      ELSIF (_Mover.NcToPlc.ModuloActPos > stGearData.rModuloSyncPosSlave + stMoveData.rDelta)
      THEN
        _nErrorId             := 667;
        _eState               := E_PROGRESS.PROGRESS_ERROR;
      END_IF
    END_IF
END_CASE
//-----------------------------------------------------------------------------
//-----------------------------------------------------------------------------
CASE _eState
OF
  E_PROGRESS.PROGRESS_BUSY:
    _eState                   := E_PROGRESS.PROGRESS_PREPARE;

    _fbPower.Override         := stMoveData.rOverride;

    _fbGearInPosCa(
        Master                := _Master, 
        Slave                 := _Mover, 
        Execute               := FALSE, 
        ContinuousUpdate      := TRUE, 
        RatioNumerator        := stGearData.rGearNumerator, 
        RatioDenumerator      := stGearData.iGearDenumerator, 

        MasterSyncPosition    := _Master.NcToPlc.ActPos 
                               + stGearData.rDeltaToMasterPos,                            // absolute position

        SlaveSyncPosition     := ABS(_Mover.NcToPlc.ModuloActTurns)*_RailLength
                               + stGearData.rModuloSyncPosSlave,                          // absolute position

        SyncStrategy          := Tc3_Mc3Definitions.MC_SYNC_STRATEGY.mcSyncStrategySlow,  // minimal movement with this strategy 
        SyncMode              := Tc3_Mc3Definitions.MC_SYNC_MODE.mcSyncModeNonModulo,     // all positions as absolute value
        MasterStartDistance   := stGearData.rMasterStartDistance,                         // if <> 0 --> master has to move before this fb does anything
        Velocity              := stMoveData.rVelo, 
        Acceleration          := stMoveData.rAcc, 
        Deceleration          := stMoveData.rAcc, 
        Jerk                  := stMoveData.rJerk, 
        Gap                   := stMoveData.rGap, 
        BufferMode            := Tc3_Mc3Definitions.MC_BUFFER_MODE.mcAborting);
END_CASE
//-----------------------------------------------------------------------------
//-----------------------------------------------------------------------------
CASE _eState
OF
  E_PROGRESS.PROGRESS_PREPARE:
    _fbGearInPosCa(
        Master                := _Master, 
        Slave                 := _Mover, 
        Execute               := TRUE, 
        ContinuousUpdate      := TRUE);

    IF _fbGearInPosCa.Error
    THEN
      _nErrorId               := _fbGearInPosCa.ErrorId;
      _eState                 := E_PROGRESS.PROGRESS_ERROR;

    ELSIF _fbGearInPosCa.CommandAborted
    THEN
      _eState                 := E_PROGRESS.PROGRESS_OCCUPIED;

    ELSIF _fbGearInPosCa.InSync
    THEN
      _eState                 := E_PROGRESS.PROGRESS_DONE;
    END_IF
END_CASE
//-----------------------------------------------------------------------------
//-----------------------------------------------------------------------------
CASE _eState
OF
  E_PROGRESS.PROGRESS_ERROR,
  E_PROGRESS.PROGRESS_DONE:
    _stInfo.nErrorId          := _nErrorId;
    _fbGearInPosCa(
        Master                := _Master, 
        Slave                 := _Mover, 
        Execute               := FALSE, 
        ContinuousUpdate      := TRUE);
END_CASE
//-----------------------------------------------------------------------------
//-----------------------------------------------------------------------------

GearInPosCa                   := _eState;
END_METHOD

METHOD GearOut : E_PROGRESS
VAR_INPUT
  Execute             : BOOL;
END_VAR
VAR_INST
  _nErrorId           : UDINT;
  _eState             : E_PROGRESS;
END_VAR
IF NOT Execute THEN _eState  := E_PROGRESS.PROGRESS_INIT; END_IF 
IF NOT Check() THEN GearOut  := E_PROGRESS.PROGRESS_ERROR; RETURN; END_IF


CASE _eState
OF
  E_PROGRESS.PROGRESS_INIT:
    IF Execute
    THEN
      _nErrorId               := 0;
      _eState                 := E_PROGRESS.PROGRESS_BUSY;
    END_IF
END_CASE
//-----------------------------------------------------------------------------
//-----------------------------------------------------------------------------
CASE _eState
OF
  E_PROGRESS.PROGRESS_BUSY:
    _eState                   := E_PROGRESS.PROGRESS_PREPARE;
    _fbGearOut(
            Slave             := _Mover, 
            Execute           := FALSE);
END_CASE
//-----------------------------------------------------------------------------
//-----------------------------------------------------------------------------
CASE _eState
OF
  E_PROGRESS.PROGRESS_PREPARE:
    _fbGearOut(
            Slave             := _Mover, 
            Execute           := TRUE);

    IF _fbGearOut.Error
    THEN
      _nErrorId               := _fbGearOut.ErrorID;
      _eState                 := E_PROGRESS.PROGRESS_ERROR;

    ELSIF (_Mover.NcToPlc.CoupleState = 0)
    THEN
      _eState                 := E_PROGRESS.PROGRESS_DONE;
    END_IF
END_CASE
//-----------------------------------------------------------------------------
//-----------------------------------------------------------------------------
CASE _eState
OF
  E_PROGRESS.PROGRESS_ERROR,
  E_PROGRESS.PROGRESS_DONE:
    _stInfo.nErrorId          := _nErrorId;
    _fbGearOut(
            Slave             := _Mover, 
            Execute           := FALSE);
END_CASE
//-----------------------------------------------------------------------------
//-----------------------------------------------------------------------------

GearOut                       := _eState;
END_METHOD

METHOD Halt : E_PROGRESS
VAR_INPUT
  Execute             : BOOL;
  stMoveData          : ST_MOVE_DATA;
END_VAR
VAR_INST
  _nErrorId           : UDINT;
  _eState             : E_PROGRESS;
END_VAR
IF NOT Execute 
THEN 
	_eState := E_PROGRESS.PROGRESS_INIT; 
END_IF 
IF NOT Check() 
THEN 
	Halt := E_PROGRESS.PROGRESS_ERROR; 
	RETURN; 
END_IF


CASE _eState
OF
  E_PROGRESS.PROGRESS_INIT:
    IF Execute
    THEN
      _nErrorId               := 0;
      _eState                 := E_PROGRESS.PROGRESS_BUSY;
    END_IF
END_CASE
//-----------------------------------------------------------------------------
//-----------------------------------------------------------------------------
CASE _eState
OF
  E_PROGRESS.PROGRESS_BUSY:
    _eState                   := E_PROGRESS.PROGRESS_PREPARE;
    _fbHalt(
            Axis              := _Mover, 
            Execute           := FALSE, 
            Deceleration      := stMoveData.rAcc, 
            Jerk              := stMoveData.rJerk, 
            BufferMode        := Tc2_MC2.MC_BufferMode.MC_Aborting);
END_CASE
//-----------------------------------------------------------------------------
//-----------------------------------------------------------------------------
CASE _eState
OF
  E_PROGRESS.PROGRESS_PREPARE:
    _fbHalt(Axis              := _Mover, 
            Execute           := TRUE, 
            Deceleration      := stMoveData.rAcc, 
            Jerk              := stMoveData.rJerk, 
            BufferMode        := Tc2_MC2.MC_BufferMode.MC_Aborting);

    IF _fbHalt.Error
    THEN
      _nErrorId               := _fbHalt.ErrorID;
      _eState                 := E_PROGRESS.PROGRESS_ERROR;

    ELSIF NOT _Mover.Status.Moving
    THEN
      _eState                 := E_PROGRESS.PROGRESS_DONE;
    END_IF
END_CASE
//-----------------------------------------------------------------------------
//-----------------------------------------------------------------------------
CASE _eState
OF
  E_PROGRESS.PROGRESS_ERROR,
  E_PROGRESS.PROGRESS_DONE:
    _stInfo.nErrorId          := _nErrorId;
    _fbHalt(
            Axis              := _Mover, 
            Execute           := FALSE);
END_CASE
//-----------------------------------------------------------------------------
//-----------------------------------------------------------------------------

Halt                          := _eState;
END_METHOD

PROPERTY LastGap : REFERENCE to lreal
SET
_rLastGap REF= LastGap;
END_SET
END_PROPERTY

PROPERTY LastPosition : REFERENCE to LREAL
SET
_rLastPosition REF= LastPosition;
END_SET
END_PROPERTY

PROPERTY Master : REFERENCE to AXIS_REF
SET
_Master REF= Master;
END_SET
END_PROPERTY

PROPERTY ModuloTurn : dint
GET
ModuloTurn := _Mover.NcToPlc.ModuloSetTurns;
END_GET
END_PROPERTY

PROPERTY Mover : REFERENCE to AXIS_REF
SET
_Mover REF= Mover;
END_SET
END_PROPERTY

PROPERTY MoverInfo : REFERENCE to ST_MOVER_INFO
SET


	_stInfo ref= MoverInfo;
END_SET
END_PROPERTY

METHOD MoveToPos : E_PROGRESS
VAR_INPUT
  Execute             : BOOL;
  stMoveData          : ST_MOVE_DATA;
END_VAR
VAR_INST
  _nErrorId           : UDINT;
  _rPos               : LREAL;
  _eState             : E_PROGRESS;
END_VAR
IF NOT Execute THEN _eState  := E_PROGRESS.PROGRESS_INIT; END_IF 
IF NOT Check() THEN MoveToPos   := E_PROGRESS.PROGRESS_ERROR; RETURN; END_IF


CASE _eState
OF
  E_PROGRESS.PROGRESS_INIT:
    IF Execute
    THEN
      _nErrorId               := 0;
      _eState                 := E_PROGRESS.PROGRESS_BUSY;
    END_IF
END_CASE
//-----------------------------------------------------------------------------
//-----------------------------------------------------------------------------
CASE _eState
OF
  E_PROGRESS.PROGRESS_BUSY:
    _eState                   := E_PROGRESS.PROGRESS_PREPARE;
    _fbPower.Override         := stMoveData.rOverride;

    _rPos                     := ABS(_Mover.NcToPlc.ModuloActTurns)* _RailLength + stMoveData.rPos;


    _rLastPosition            := _rPos;
    //_rLastGap                 := stMoveData.rGap;

    _fbMoveAbs(
            Axis              := _Mover, 
            Execute           := FALSE, 
            Position          := _rPos, 
            Velocity          := stMoveData.rVelo, 
            Acceleration      := stMoveData.rAcc, 
            Deceleration      := stMoveData.rAcc, 
            Jerk              := stMoveData.rJerk, 
            BufferMode        := Tc2_MC2.MC_BufferMode.MC_Aborting);
END_CASE
//-----------------------------------------------------------------------------
//-----------------------------------------------------------------------------
CASE _eState
OF
  E_PROGRESS.PROGRESS_PREPARE:
    _fbMoveAbs(
            Axis              := _Mover, 
            Execute           := TRUE, 
            Position          := _rPos, 
            Velocity          := stMoveData.rVelo, 
            Acceleration      := stMoveData.rAcc, 
            Deceleration      := stMoveData.rAcc, 
            Jerk              := stMoveData.rJerk, 
            BufferMode        := Tc2_MC2.MC_BufferMode.MC_Aborting);

    IF _fbMoveAbs.Error
    THEN
      _nErrorId               := _fbMoveAbs.ErrorId;
      _eState                 := E_PROGRESS.PROGRESS_ERROR;

    ELSIF _fbMoveAbs.Active OR 
          _fbMoveAbs.Done
		THEN
      _eState                 := E_PROGRESS.PROGRESS_WORKING;
    END_IF
END_CASE
//-----------------------------------------------------------------------------
//-----------------------------------------------------------------------------
CASE _eState
OF
  E_PROGRESS.PROGRESS_WORKING:
    _fbMoveAbs(
          Axis              := _Mover);

    IF _fbMoveAbs.Error
    THEN
      _nErrorId             := _fbMoveAbs.ErrorId;
      _eState               := E_PROGRESS.PROGRESS_ERROR;

    ELSIF (_Mover.NcToPlc.ActPos > _fbMoveAbs.Position - stMoveData.rDelta) AND
          (_Mover.NcToPlc.ActPos < _fbMoveAbs.Position + stMoveData.rDelta)
    THEN
      IF NOT _Mover.Status.Moving
      THEN
        _eState               := E_PROGRESS.PROGRESS_DONE;
      END_IF
    END_IF
END_CASE
//-----------------------------------------------------------------------------
//-----------------------------------------------------------------------------
CASE _eState
OF
  E_PROGRESS.PROGRESS_ERROR,
  E_PROGRESS.PROGRESS_DONE:
    _stInfo.nErrorId          := _nErrorId;
    _fbMoveAbs( 
            Axis              := _Mover, 
            Execute           := FALSE);
END_CASE
//-----------------------------------------------------------------------------
//-----------------------------------------------------------------------------

MoveToPos                   := _eState;
END_METHOD

METHOD MoveToPosCa : E_PROGRESS
VAR_INPUT
  Execute             : BOOL;
  stMoveData          : ST_MOVE_DATA;
END_VAR
VAR_INST
  _nErrorId           : UDINT;
  _rPos               : LREAL;
  _eState             : E_PROGRESS;
END_VAR
IF NOT Execute THEN _eState  := E_PROGRESS.PROGRESS_INIT; END_IF 
IF NOT Check() THEN MoveToPosCa   := E_PROGRESS.PROGRESS_ERROR; RETURN; END_IF


CASE _eState
OF
  E_PROGRESS.PROGRESS_INIT:
    IF Execute
    THEN
      _nErrorId               := 0;
      _eState                 := E_PROGRESS.PROGRESS_BUSY;
    END_IF
END_CASE
//-----------------------------------------------------------------------------
//-----------------------------------------------------------------------------
CASE _eState
OF
  E_PROGRESS.PROGRESS_BUSY:
    _eState                   := E_PROGRESS.PROGRESS_PREPARE;
    _fbPower.Override         := stMoveData.rOverride;

    _rPos                     := ABS(_Mover.NcToPlc.ModuloActTurns)* _RailLength + stMoveData.rPos;


    _rLastPosition            := _rPos;
    _rLastGap                 := stMoveData.rGap;

    _fbMoveAbsCa( 
            Axis              := _Mover, 
            Execute           := FALSE, 
            ContinuousUpdate  := TRUE, 
            Position          := _rPos,
            Velocity          := stMoveData.rVelo, 
            Acceleration      := stMoveData.rAcc, 
            Deceleration      := stMoveData.rAcc, 
            Jerk              := stMoveData.rJerk, 
            Gap               := stMoveData.rGap, 
            BufferMode        := Tc3_Mc3Definitions.MC_BUFFER_MODE.mcAborting);
END_CASE
//-----------------------------------------------------------------------------
//-----------------------------------------------------------------------------
CASE _eState
OF
  E_PROGRESS.PROGRESS_PREPARE:
    _fbMoveAbsCa( 
            Axis              := _Mover, 
            Execute           := TRUE, 
            ContinuousUpdate  := TRUE, 
            Position          := _rPos,
            Velocity          := stMoveData.rVelo, 
            Acceleration      := stMoveData.rAcc, 
            Deceleration      := stMoveData.rAcc, 
            Jerk              := stMoveData.rJerk, 
            Gap               := stMoveData.rGap, 
            BufferMode        := Tc3_Mc3Definitions.MC_BUFFER_MODE.mcAborting);

    IF _fbMoveAbsCa.Error
    THEN
      _nErrorId               := _fbMoveAbsCa.ErrorId;
      _eState                 := E_PROGRESS.PROGRESS_ERROR;

    ELSIF _fbMoveAbsCa.Active OR 
          _fbMoveAbsCa.Done
		THEN
      _eState                 := E_PROGRESS.PROGRESS_WORKING;
    END_IF
END_CASE
//-----------------------------------------------------------------------------
//-----------------------------------------------------------------------------
CASE _eState
OF
  E_PROGRESS.PROGRESS_WORKING:
    _fbMoveAbsCa(
          Axis              := _Mover);

    IF _fbMoveAbsCa.Error
    THEN
      _nErrorId             := _fbMoveAbsCa.ErrorId;
      _eState               := E_PROGRESS.PROGRESS_ERROR;

    ELSIF (_Mover.NcToPlc.ActPos > _fbMoveAbsCa.Position - stMoveData.rDelta) AND
          (_Mover.NcToPlc.ActPos < _fbMoveAbsCa.Position + stMoveData.rDelta)
    THEN
      IF NOT _Mover.Status.Moving
      THEN
        _eState               := E_PROGRESS.PROGRESS_DONE;
      END_IF
    END_IF
END_CASE
//-----------------------------------------------------------------------------
//-----------------------------------------------------------------------------
CASE _eState
OF
  E_PROGRESS.PROGRESS_ERROR,
  E_PROGRESS.PROGRESS_DONE:
    _stInfo.nErrorId          := _nErrorId;
    _fbMoveAbsCa( 
            Axis              := _Mover, 
            Execute           := FALSE);
END_CASE
//-----------------------------------------------------------------------------
//-----------------------------------------------------------------------------

MoveToPosCa                   := _eState;
END_METHOD

PROPERTY RailLength : LREAL
GET
RailLength := _RailLength;
END_GET
SET
_RailLength := RailLength;
END_SET
END_PROPERTY

METHOD Reset : E_PROGRESS
VAR_INPUT
  Execute             : BOOL;
END_VAR
VAR_INST
  _nErrorId           : UDINT;
  _eState             : E_PROGRESS;
END_VAR
IF NOT Execute THEN _eState  := E_PROGRESS.PROGRESS_INIT; END_IF 
IF NOT Check() THEN Reset    := E_PROGRESS.PROGRESS_ERROR; RETURN; END_IF


CASE _eState
OF
  E_PROGRESS.PROGRESS_INIT:
    IF Execute
    THEN
      _stInfo.nErrorId        :=
      _nErrorId               := 0;
      _eState                 := E_PROGRESS.PROGRESS_BUSY;
    END_IF
END_CASE
//-----------------------------------------------------------------------------
//-----------------------------------------------------------------------------
CASE _eState
OF
  E_PROGRESS.PROGRESS_BUSY:
    _eState                   := E_PROGRESS.PROGRESS_PREPARE;
    _fbReset(
            Axis              := _Mover, 
            Execute           := FALSE);
END_CASE
//-----------------------------------------------------------------------------
//-----------------------------------------------------------------------------
CASE _eState
OF
  E_PROGRESS.PROGRESS_PREPARE:
    _fbReset(
            Axis              := _Mover, 
            Execute           := TRUE);

    IF _fbReset.Error
    THEN
      _nErrorId               := _fbReset.ErrorID;
      _eState                 := E_PROGRESS.PROGRESS_ERROR;

    ELSIF NOT _Mover.Status.Moving
    THEN
      _eState                 := E_PROGRESS.PROGRESS_DONE;
    END_IF
END_CASE
//-----------------------------------------------------------------------------
//-----------------------------------------------------------------------------
CASE _eState
OF
  E_PROGRESS.PROGRESS_ERROR,
  E_PROGRESS.PROGRESS_DONE:
    _stInfo.nErrorId          := _nErrorId;
    _fbReset(
            Axis              := _Mover, 
            Execute           := FALSE);
			
	_bError := FALSE;		
END_CASE
//-----------------------------------------------------------------------------
//-----------------------------------------------------------------------------

Reset                         := _eState;
END_METHOD

METHOD SendToAbsPosCa : E_PROGRESS
VAR_INPUT
  Execute             : BOOL;
  stMoveData          : ST_MOVE_DATA;
END_VAR
VAR_INST
  _nErrorId           : UDINT;
  _rPos               : LREAL;
  _rStart             : LREAL;
  _eState             : E_PROGRESS;
END_VAR
IF NOT Execute THEN _eState  := E_PROGRESS.PROGRESS_INIT; END_IF 
IF NOT Check() THEN SendToAbsPosCa   := E_PROGRESS.PROGRESS_ERROR; RETURN; END_IF


CASE _eState
OF
  E_PROGRESS.PROGRESS_INIT:
    IF Execute
    THEN
      _nErrorId               := 0;
      _rStart                 := _Mover.NcToPlc.ActPos;

      _eState                 := E_PROGRESS.PROGRESS_BUSY;
    END_IF
END_CASE
//-----------------------------------------------------------------------------
//-----------------------------------------------------------------------------
CASE _eState
OF
  E_PROGRESS.PROGRESS_BUSY:
    _eState                   := E_PROGRESS.PROGRESS_PREPARE;
    _fbPower.Override         := stMoveData.rOverride;

    _rPos                     := stMoveData.rPos;
	
    _rLastPosition            := _rPos;
    _rLastGap                 := stMoveData.rGap;

    _fbMoveAbsCa( 
            Axis              := _Mover, 
            Execute           := FALSE, 
            ContinuousUpdate  := TRUE, 
            Position          := _rPos,
            Velocity          := stMoveData.rVelo, 
            Acceleration      := stMoveData.rAcc, 
            Deceleration      := stMoveData.rAcc, 
            Jerk              := stMoveData.rJerk, 
            Gap               := stMoveData.rGap, 
            BufferMode        := Tc3_Mc3Definitions.MC_BUFFER_MODE.mcAborting);
END_CASE
//-----------------------------------------------------------------------------
//-----------------------------------------------------------------------------
CASE _eState
OF
  E_PROGRESS.PROGRESS_PREPARE:
    _fbMoveAbsCa( 
            Axis              := _Mover, 
            Execute           := TRUE, 
            ContinuousUpdate  := TRUE, 
            Position          := _rPos,
            Velocity          := stMoveData.rVelo, 
            Acceleration      := stMoveData.rAcc, 
            Deceleration      := stMoveData.rAcc, 
            Jerk              := stMoveData.rJerk, 
            Gap               := stMoveData.rGap, 
            BufferMode        := Tc3_Mc3Definitions.MC_BUFFER_MODE.mcAborting);

    IF _fbMoveAbsCa.Error
    THEN
      _nErrorId               := _fbMoveAbsCa.ErrorId;
      _eState                 := E_PROGRESS.PROGRESS_ERROR;

    ELSIF _fbMoveAbsCa.Active
    THEN
      _eState                 := E_PROGRESS.PROGRESS_WORKING;
    END_IF
END_CASE
//-----------------------------------------------------------------------------
//-----------------------------------------------------------------------------
CASE _eState
OF
  E_PROGRESS.PROGRESS_WORKING:
    _fbMoveAbsCa(
            Axis              := _Mover);

    IF _fbMoveAbsCa.Error
    THEN
      _nErrorId               := _fbMoveAbsCa.ErrorId;
      _eState                 := E_PROGRESS.PROGRESS_ERROR;

    ELSIF (_Mover.NcToPlc.ActPos > _rStart + stMoveData.rDistance)
    THEN
      _eState                 := E_PROGRESS.PROGRESS_DONE;
    END_IF
END_CASE
//-----------------------------------------------------------------------------
//-----------------------------------------------------------------------------
CASE _eState
OF
  E_PROGRESS.PROGRESS_ERROR,
  E_PROGRESS.PROGRESS_DONE:
    _stInfo.nErrorId          := _nErrorId;
    _fbMoveAbsCa( 
            Axis              := _Mover, 
            Execute           := FALSE);
END_CASE
//-----------------------------------------------------------------------------
//-----------------------------------------------------------------------------

SendToAbsPosCa                := _eState;
END_METHOD

METHOD SendToModuloPosCa : E_PROGRESS
VAR_INPUT
  Execute             : BOOL;
  stMoveData          : ST_MOVE_DATA;
END_VAR
VAR_INST
  _nErrorId           : UDINT;
  _rPos               : LREAL;
  _rStart             : LREAL;
  _eState             : E_PROGRESS;
END_VAR
IF NOT Execute THEN _eState  := E_PROGRESS.PROGRESS_INIT; END_IF 
IF NOT Check() THEN SendToModuloPosCa   := E_PROGRESS.PROGRESS_ERROR; RETURN; END_IF


CASE _eState
OF
  E_PROGRESS.PROGRESS_INIT:
    IF Execute
    THEN
      _nErrorId               := 0;
      _rStart                 := _Mover.NcToPlc.ActPos;

      _eState                 := E_PROGRESS.PROGRESS_BUSY;
    END_IF
END_CASE
//-----------------------------------------------------------------------------
//-----------------------------------------------------------------------------
CASE _eState
OF
  E_PROGRESS.PROGRESS_BUSY:
    _eState                   := E_PROGRESS.PROGRESS_PREPARE;
    _fbPower.Override         := stMoveData.rOverride;

    _rPos                     := ABS(_Mover.NcToPlc.ModuloActTurns)* _RailLength + stMoveData.rPos;
	
    _rLastPosition            := _rPos;
    _rLastGap                 := stMoveData.rGap;

    _fbMoveAbsCa( 
            Axis              := _Mover, 
            Execute           := FALSE, 
            ContinuousUpdate  := TRUE, 
            Position          := _rPos,
            Velocity          := stMoveData.rVelo, 
            Acceleration      := stMoveData.rAcc, 
            Deceleration      := stMoveData.rAcc, 
            Jerk              := stMoveData.rJerk, 
            Gap               := stMoveData.rGap, 
            BufferMode        := Tc3_Mc3Definitions.MC_BUFFER_MODE.mcAborting);
END_CASE
//-----------------------------------------------------------------------------
//-----------------------------------------------------------------------------
CASE _eState
OF
  E_PROGRESS.PROGRESS_PREPARE:
    _fbMoveAbsCa( 
            Axis              := _Mover, 
            Execute           := TRUE, 
            ContinuousUpdate  := TRUE, 
            Position          := _rPos,
            Velocity          := stMoveData.rVelo, 
            Acceleration      := stMoveData.rAcc, 
            Deceleration      := stMoveData.rAcc, 
            Jerk              := stMoveData.rJerk, 
            Gap               := stMoveData.rGap, 
            BufferMode        := Tc3_Mc3Definitions.MC_BUFFER_MODE.mcAborting);

    IF _fbMoveAbsCa.Error
    THEN
      _nErrorId               := _fbMoveAbsCa.ErrorId;
      _eState                 := E_PROGRESS.PROGRESS_ERROR;

    ELSIF _fbMoveAbsCa.Active
    THEN
      _eState                 := E_PROGRESS.PROGRESS_WORKING;
    END_IF
END_CASE
//-----------------------------------------------------------------------------
//-----------------------------------------------------------------------------
CASE _eState
OF
  E_PROGRESS.PROGRESS_WORKING:
    _fbMoveAbsCa(
            Axis              := _Mover);

    IF _fbMoveAbsCa.Error
    THEN
      _nErrorId               := _fbMoveAbsCa.ErrorId;
      _eState                 := E_PROGRESS.PROGRESS_ERROR;

    ELSIF (_Mover.NcToPlc.ActPos > _rStart + stMoveData.rDistance)
    THEN
      _eState                 := E_PROGRESS.PROGRESS_DONE;
    END_IF
END_CASE
//-----------------------------------------------------------------------------
//-----------------------------------------------------------------------------
CASE _eState
OF
  E_PROGRESS.PROGRESS_ERROR,
  E_PROGRESS.PROGRESS_DONE:
    _stInfo.nErrorId          := _nErrorId;
    _fbMoveAbsCa( 
            Axis              := _Mover, 
            Execute           := FALSE);
END_CASE
//-----------------------------------------------------------------------------
//-----------------------------------------------------------------------------

SendToModuloPosCa                   := _eState;
END_METHOD

END_FUNCTION_BLOCK

// ---- XTS/XtsStation/fb_Station.TcPOU
//---------------------------------------------------------------------------------------------------------------
//
//  HAUD 2023.03.07
//
//  TR06
//  - XTS_TRAINING
//  - example project for setting up transport layer
//
//
//  fb_Station
//  - handshake with extern control for mover transport through station
//
//---------------------------------------------------------------------------------------------------------------
// This SOFTWARE is provided as an Exemple by THE PROVIDER "as is" and "with all faults." THE PROVIDER makes no 
// representations or warranties of any kind concerning the safety, suitability, lack of viruses, inaccuracies, 
// typographical errors, or other harmful components of this SOFTWARE. There are inherent dangers in the use of 
// any software, and you are solely responsible for determining whether this SOFTWARE is compatible with your 
// equipment and other software installed on your equipment. You are also solely responsible for the protection 
// of your equipment and backup of your data, and THE PROVIDER will not be liable for any damages you may suffer 
// in connection with using, modifying, or distributing this SOFTWARE.
//---------------------------------------------------------------------------------------------------------------
FUNCTION_BLOCK fb_Station IMPLEMENTS I_XtsTransport_Station
VAR
  _nStationId                 : UINT;         // why is Gamora?

  _sState                     : STRING(255);  // additional output for Check()

  // pointer to all stations
  _stCtrl                     : POINTER TO ARRAY[1..MAX_STATION]  OF ST_STATION_CTRL;
  _stState                    : POINTER TO ARRAY[1..MAX_STATION]  OF ST_STATION_STATE;

  // local copy of me
  _stStationCtrl              : ST_STATION_CTRL;
  _stStationState             : ST_STATION_STATE;

  _ItfStation                 : POINTER TO ARRAY[1..MAX_STATION]  OF I_Station_LinkedList;  // access to all stations lists
  _ItfMover                   : POINTER TO ARRAY[1..MAX_MOVER]    OF I_XtsTransport_Mover;  // access to mover methods

  // station related data
  _rMoverOffset               : POINTER TO ARRAY[1..MAX_STATION]  OF T_NEST_OFFSET;         // static offsets for station

  _stParameter                : POINTER TO ARRAY[1..MAX_STATION]  OF ST_STATION_PARAMETER;  // station parameter (where, how fast, how many stops)

  _Mover                      : POINTER TO ARRAY[1..MAX_MOVER]    OF AXIS_REF;              // read from AXIS_REF

  // linked list result struct
  _stListEnter,
  _stListTarget,
  _stListDelete               : ST_STATION_LIST_RESULT;   // struct with result and ticket data

  _stMoverDataSend,
  _stMoverData                : ST_STATION_MOVER_DATA;    // mover ticket data

  _stMoveData                 : ST_MOVE_DATA;             // position and dynamic constraints of movement

  // work vars
  _bInitList                  : BOOL;

  _Result                     : E_PROGRESS;

  _eState                     : E_PROGRESS;

  _nNest,
  _nMoverDetected,
  _nMoverInStation,
  _nTargetStation,
  _ix                         : UINT;

  _rWork                      : LREAL;
  _rModActPosFetch            : LREAL;

  _eFatalError                : E_STATION_STATE;
END_VAR

METHOD PRIVATE Check : BOOL
VAR_INPUT
END_VAR
IF NOT (_nStationId > 0) OR
       (_nStationId > MAX_STATION)
THEN
  _sState                     := 'invalid nStationId';
  RETURN;
END_IF

IF NOT (_stCtrl  <> 0)
THEN
  _sState                     := '_stCtrl: missing pointer';
  RETURN;
END_IF

IF NOT (_stState <> 0)
THEN
  _sState                     := '_stState: missing pointer';
  RETURN;
END_IF

IF NOT (_ItfStation <> 0)
THEN
  _sState                     := '_ItfStation: missing interface';
  RETURN;
END_IF

IF NOT (_ItfMover <> 0)
THEN
  _sState                     := '_ItfMover: missing interface';
  RETURN;
END_IF

IF NOT (_rMoverOffset  <> 0)
THEN
  _sState                     := '_rMoverOffset: missing pointer';
  RETURN;
END_IF

IF NOT (_stParameter  <> 0)
THEN
  _sState                     := '_stParameter: missing pointer';
  RETURN;
END_IF

IF NOT (_Mover  <> 0)
THEN
  _sState                     := '_Mover: missing pointer';
  RETURN;
END_IF


_sState                       := 'CHECK_DONE';
Check                         := TRUE;
END_METHOD

PROPERTY Ctrl : pointer to ARRAY[1..MAX_STATION] OF ST_STATION_CTRL
SET
_stCtrl := Ctrl;
END_SET
END_PROPERTY

METHOD Cycle
// check pointer and interface
IF NOT Check() THEN RETURN; END_IF

// direct from interface
CASE _stCtrl^[_nStationId].eCmd
OF
  E_STATION_CTRL.STATION_INIT:      // commanded init from cyclic interface
    Init();
    RETURN;


  E_STATION_CTRL.STATION_DISABLE:   // commanded disable from cyclic interface
    CASE _stStationState.eState
    OF
      E_STATION_STATE.STATION_INIT,
      E_STATION_STATE.STATION_DISABLE:
        // disable station when no mover is handled
        _stStationState.eState        := E_STATION_STATE.STATION_DISABLE;
    END_CASE
END_CASE

//-----------------------------------------------------------------------------
// copy ctrl to local
//-----------------------------------------------------------------------------
_stStationCtrl                        := _stCtrl^[_nStationId];
//-----------------------------------------------------------------------------
//-----------------------------------------------------------------------------
CASE _stStationState.eState
OF
  E_STATION_STATE.STATION_NO_INIT:    // startup state in first PLC cycle, init linked list required
    IF NOT _bInitList
    THEN
      _bInitList                      := _ItfStation^[_nStationId].InitList();
    END_IF
    _stStationState.eState            := E_STATION_STATE.STATION_INIT;

  E_STATION_STATE.STATION_INIT:       // switch state as reserve for anything you might add here
    _stStationState.nMoverId          := 0;
    _stStationState.eState            := E_STATION_STATE.STATION_DISABLE;
END_CASE
//-----------------------------------------------------------------------------
//-----------------------------------------------------------------------------
CASE _stStationState.eState
OF
  E_STATION_STATE.STATION_DISABLE:    // end state after first PLC cycle startup; wait state after commanded disable
    IF (_stStationCtrl.eCmd = E_STATION_CTRL.STATION_ENABLE)
    THEN
      _stStationState.eState          := E_STATION_STATE.STATION_ENABLE;
    END_IF


  E_STATION_STATE.STATION_ENABLE:     // double check commanded enable and clear work vars
    IF (_stStationCtrl.eCmd = E_STATION_CTRL.STATION_ENABLE)
    THEN
      memset(ADR(_stListEnter),    0, SIZEOF(_stListEnter));

      _eState                         := E_PROGRESS.PROGRESS_INIT;  // work var for nested case
      _stStationState.eState          := E_STATION_STATE.STATION_DETECT_MOVER;
    END_IF


  E_STATION_STATE.STATION_DETECT_MOVER:// wait state for mover detection
    CASE _eState
    OF
      E_PROGRESS.PROGRESS_INIT:
        IF (_stStationCtrl.eCmd = E_STATION_CTRL.STATION_DISABLE) // check for commanded disable
        THEN
          _stStationState.eState      := E_STATION_STATE.STATION_DISABLE; // go back and wait, no matter the queue

        ELSIF (_ItfStation^[_nStationId].Count > 0)
        THEN
          // someone entered something in my list
          _stListEnter                := _ItfStation^[_nStationId].GetHead();
          _eState                     := E_PROGRESS.PROGRESS_BUSY;
        END_IF
    END_CASE
    CASE _eState
    OF
      E_PROGRESS.PROGRESS_BUSY:
        IF (_stListEnter.wState = 0)  // GetHead() without error
        THEN
          // list is giving head as result
          _stMoverData                := _stListEnter.stData; // copy ticket from list result
          _eState                     := E_PROGRESS.PROGRESS_PREPARE;
        ELSE
          // the thing that must not be: GetHead() with error
          _stStationState.eState      := E_STATION_STATE.STATION_ERROR_LIST_GET_HEAD_FAULT;
        END_IF
    END_CASE
    CASE _eState
    OF
      E_PROGRESS.PROGRESS_PREPARE:    // check ticket (list entry)
        // check target assignement
        IF NOT (_stMoverData.nTargetStation = _nStationId)
        THEN
          // for whom the mover calls
          // wrong address, right mover?
          _stStationState.eState      := E_STATION_STATE.STATION_ERROR_LIST_STATION_ID_WRONG;
        ELSE
          // it's a me
          _nMoverDetected             := _stMoverData.nMoverId;

          IF (_nMoverDetected < 1) OR
             (_nMoverDetected > MAX_MOVER)
          THEN
            // out of range the mover must not be
            _stStationState.eState    := E_STATION_STATE.STATION_ERROR_LIST_MOVER_ID_INVALID;
          ELSE
            memset(ADR(_stListDelete),   0, SIZEOF(_stListDelete)); // clear work var
            _eState                   := E_PROGRESS.PROGRESS_INIT;

            // prepare station state for new mover
            _stStationState.nMoverId  := TO_USINT(_nMoverDetected); // who has arrived
            _stStationState.nMask     := _stMoverData.nMask;        // how many stops have to be made
            _stStationState.eState    := E_STATION_STATE.STATION_MOVER_ENTER; // go ask for permission to enter
          END_IF
        END_IF
    END_CASE
END_CASE
//-----------------------------------------------------------------------------
//-----------------------------------------------------------------------------
CASE _stStationState.eState
OF
  E_STATION_STATE.STATION_MOVER_ENTER:  // requesting permission for mover to enter station
    CASE _eState
    OF
      E_PROGRESS.PROGRESS_INIT:
        IF (_stStationCtrl.eCmd = E_STATION_CTRL.STATION_DISABLE)
        THEN
          _stStationState.eState      := E_STATION_STATE.STATION_DISABLE;
        ELSE
          IF (_stStationCtrl.eCmd = E_STATION_CTRL.STATION_MOVER_ENTER)   // mover may enter station now
          THEN
            _nNest                    := 1; // default nest
            _eState                   := E_PROGRESS.PROGRESS_BUSY;

            FOR _ix := 1 TO _stParameter^[_nStationId].nConfiguredStopCount
            DO
              IF GetBitWord(_stMoverData.nMask, _ix-1)
              THEN
                _nNest                := _ix;
                EXIT;
              END_IF
            END_FOR

          ELSIF (_stStationCtrl.eCmd = E_STATION_CTRL.STATION_MOVER_SEND) // control decided otherwise, mover shall be sent away
          THEN
            _stStationState.eState    := E_STATION_STATE.STATION_MOVER_OUT;
          END_IF
        END_IF
    END_CASE
    CASE _eState
    OF
      E_PROGRESS.PROGRESS_BUSY:
        MoveData();

        // check if infeed movement has to cross modulo turn
        _rModActPosFetch            := _Mover^[_stMoverData.nMoverId].NcToPlc.ModuloActPos;

        IF (_rModActPosFetch > _stMoveData.rPos + _stParameter^[_nStationId].rReleaseDistance)
        THEN
          _stMoveData.rPos          := _stMoveData.rPos + TO_REAL(_ItfMover^[_stMoverData.nMoverId].RailLength);
        END_IF

        _stStationState.eState      := E_STATION_STATE.STATION_MOVER_IN_TARGET;
    END_CASE
END_CASE
//-----------------------------------------------------------------------------
//-----------------------------------------------------------------------------
CASE _stStationState.eState
OF
  E_STATION_STATE.STATION_MOVER_IN_TARGET:
    _Result := _ItfMover^[_stMoverData.nMoverId].MoveToPosCa(TRUE, _stMoveData);

    IF (_Result = E_PROGRESS.PROGRESS_DONE)
    THEN
      // mother! has arrived
      _ItfMover^[_stMoverData.nMoverId].MoveToPosCa(FALSE, _stMoveData);

      _stStationState.eState          := E_STATION_STATE.STATION_PROCESS_START;
    ELSE
      IF (_Result = E_PROGRESS.PROGRESS_ERROR)
      THEN
        _ItfMover^[_stMoverData.nMoverId].MoveToPosCa(FALSE, _stMoveData);
        _stStationState.eState        := E_STATION_STATE.STATION_ERROR_INFEED_ERROR;
      END_IF 
    END_IF
END_CASE
//-----------------------------------------------------------------------------
//-----------------------------------------------------------------------------
CASE _stStationState.eState
OF
  E_STATION_STATE.STATION_PROCESS_START:
    IF (_stStationCtrl.eCmd = E_STATION_CTRL.STATION_PROCESS_START) OR  // double handshake, your choice
       (_stStationCtrl.eCmd = E_STATION_CTRL.STATION_PROCESS_DONE)      // single handshake, your choice
    THEN
      // clear bit in mask when started/done
      _stStationState.nMask           := TO_USINT(DelBitWord(TO_WORD(_stStationState.nMask), _nNest-1));
      _stStationState.eState          := E_STATION_STATE.STATION_PROCESS_DONE;
    END_IF
END_CASE
//-----------------------------------------------------------------------------
//-----------------------------------------------------------------------------
CASE _stStationState.eState
OF
  E_STATION_STATE.STATION_PROCESS_DONE:
    IF (_stStationCtrl.eCmd = E_STATION_CTRL.STATION_PROCESS_DONE)
    THEN
      _stStationState.eState          := E_STATION_STATE.STATION_CHECK;
    END_IF
END_CASE
//-----------------------------------------------------------------------------
//-----------------------------------------------------------------------------
CASE _stStationState.eState
OF
  E_STATION_STATE.STATION_CHECK:
    IF (_stStationState.nMask = 0)
    THEN
      // mover has to leave
      _stStationState.eState          := E_STATION_STATE.STATION_MOVER_OUT;

    ELSE
      // more work to do
      _stStationState.eState          := E_STATION_STATE.STATION_CHECK_NEST;

      FOR _ix := 1 TO _stParameter^[_nStationId].nConfiguredStopCount
      DO
        IF GetBitWord(_stStationState.nMask, _ix-1)
        THEN
          _nNest                      := _ix;
          EXIT;
        END_IF
      END_FOR
    END_IF
END_CASE
//-----------------------------------------------------------------------------
//-----------------------------------------------------------------------------
CASE _stStationState.eState
OF
  E_STATION_STATE.STATION_CHECK_NEST:
    MoveData();
    _stStationState.eState            := E_STATION_STATE.STATION_MOVER_IN_TARGET;
END_CASE
//-----------------------------------------------------------------------------
//-----------------------------------------------------------------------------
CASE _stStationState.eState
OF
  E_STATION_STATE.STATION_MOVER_OUT:
    IF (_stStationCtrl.eCmd = E_STATION_CTRL.STATION_MOVER_OUT)
    THEN
      IF (_stStationCtrl.nTargetStation < 1) OR  
         (_stStationCtrl.nTargetStation > MAX_STATION)
      THEN
        _stStationState.eState        := STATION_ERROR_OUTFEED_TARGET_INVALID;
      ELSE
        _stListDelete                 := _ItfStation^[_nStationId].RemoveHeadValue();

        IF (_stListDelete.wState <> 0)
        THEN
          _stStationState.eState      := E_STATION_STATE.STATION_ERROR_LIST_REMOVE_HEAD_FAULT;
        ELSE
          memset(ADR(_stListTarget),   0, SIZEOF(_stListTarget));

          MoverOut();
          _stStationState.eState      := E_STATION_STATE.STATION_MOVER_RELEASE;
        END_IF
      END_IF
    END_IF
END_CASE
//-----------------------------------------------------------------------------
//-----------------------------------------------------------------------------
CASE _stStationState.eState
OF
  E_STATION_STATE.STATION_MOVER_RELEASE:
    _Result                           := _ItfMover^[_stMoverDataSend.nMoverId].SendToModuloPosCa(TRUE, _stMoveData);

    IF (_Result = E_PROGRESS.PROGRESS_DONE)
    THEN
      // add entry in target station list
      _stListTarget                   := _ItfStation^[_stMoverDataSend.nTargetStation].AddTailValue(_stMoverDataSend);

      IF (_stListTarget.wState <> 0)
      THEN
        _stStationState.eState        := STATION_ERROR_LIST_ADD_TAIL_FAULT;
      ELSE
        MoverOut();
        _stStationState.eState        := E_STATION_STATE.STATION_MOVER_GONE;
      END_IF
    END_IF
END_CASE
//-----------------------------------------------------------------------------
//-----------------------------------------------------------------------------
CASE _stStationState.eState
OF
  E_STATION_STATE.STATION_MOVER_GONE:
    _ItfMover^[_stMoverDataSend.nMoverId].SendToModuloPosCa(FALSE, 
                                                      _stMoveData);

    memset(ADR(_stMoverData),  0, SIZEOF(_stMoverData));

    _stStationState.nMask             := 0;
    _stStationState.nMoverId          := 0;

    IF (_stStationCtrl.eCmd = E_STATION_CTRL.STATION_MOVER_GONE)
    THEN
      _stStationState.eState          := E_STATION_STATE.STATION_INIT;
    END_IF
END_CASE
//-----------------------------------------------------------------------------
//-----------------------------------------------------------------------------
_sState                               := TO_STRING(_stStationState.eState);
//-----------------------------------------------------------------------------
// Errors
//-----------------------------------------------------------------------------
CASE _stStationState.eState
OF
  E_STATION_STATE.STATION_ERROR_LIST_STATION_ID_WRONG:
    IF (_stStationCtrl.eCmd = E_STATION_CTRL.STATION_MOVER_OUT)
    THEN
      _nMoverDetected                 := _stMoverData.nMoverId;

      IF (_nMoverDetected < 1) OR
         (_nMoverDetected > MAX_MOVER)
      THEN
        // this MUST NOT happen
        _stStationState.eState        := E_STATION_STATE.STATION_ERROR_LIST_MOVER_ID_INVALID;
      ELSE
        // not for station; send mover out
        _stStationState.eState          := E_STATION_STATE.STATION_MOVER_OUT;
      END_IF

    ELSIF (_stStationCtrl.eCmd = E_STATION_CTRL.STATION_MOVER_ENTER)
    THEN
      // override wrong TargetStationId in List; start infeed of mover

      _nMoverDetected                 := _stMoverData.nMoverId;

      IF (_nMoverDetected < 1) OR
         (_nMoverDetected > MAX_MOVER)
      THEN
        // this MUST NOT happen
        _stStationState.eState        := E_STATION_STATE.STATION_ERROR_LIST_MOVER_ID_INVALID;
      ELSE
        _eState                       := E_PROGRESS.PROGRESS_INIT;
        _stStationState.nMoverId      := TO_USINT(_nMoverDetected);
        _stStationState.nMask         := _stMoverData.nMask;
        _stStationState.eState        := E_STATION_STATE.STATION_MOVER_ENTER;
      END_IF

    END_IF

  E_STATION_STATE.STATION_ERROR_OUTFEED_TARGET_INVALID:
    // wait here until valid target is detected
    IF NOT (_stStationCtrl.nTargetStation < 1) AND  
       NOT (_stStationCtrl.nTargetStation > MAX_STATION)
    THEN
      _stStationState.eState          := E_STATION_STATE.STATION_MOVER_OUT;
    END_IF


  E_STATION_STATE.STATION_ERROR_LIST_GET_HEAD_FAULT,
  E_STATION_STATE.STATION_ERROR_LIST_REMOVE_HEAD_FAULT,
  E_STATION_STATE.STATION_ERROR_LIST_ADD_TAIL_FAULT,
  E_STATION_STATE.STATION_ERROR_LIST_MOVER_ID_INVALID,
  E_STATION_STATE.STATION_ERROR_INFEED_ERROR:
    // yes, but why?
    // cannot be fixed by ctrl
    _eFatalError                      := _stStationState.eState;
    _stStationState.eState            := E_STATION_STATE.STATION_ERROR_FATAL;

  E_STATION_STATE.STATION_ERROR_FATAL:
    // write to string for debugging
    _sState                           := concat(TO_STRING(_stStationState.eState), ': ');
    _sState                           := concat(_sState, TO_STRING(_eFatalError));
END_CASE


_stStationState.nQueue                := TO_USINT(_ItfStation^[_nStationId].Count);
_stState^[_nStationId]                := _stStationState;
END_METHOD

METHOD PUBLIC DelBitWord : WORD
VAR_INPUT
  inVal   : WORD;
  bitNo   : DINT;
END_VAR
VAR
  wConst : WORD := 1;
END_VAR
IF ( inVal AND SHL( wConst,bitNo MOD 16 ) ) > 0 THEN
  DelBitWord := inVal XOR (SHL( wConst,bitNo MOD 16 ));
ELSE
  DelBitWord := inVal;
END_IF
END_METHOD

METHOD PUBLIC GetBitWord : BOOL
VAR_INPUT
  inVal   : WORD;
  bitNo   : DINT;
END_VAR
VAR
  wConst : WORD := 1;
END_VAR
IF ( inVal AND SHL( wConst,DINT_TO_SINT(bitNo) MOD 16 ) ) > 0
THEN
  GetBitWord := TRUE;
ELSE
  GetBitWord := FALSE;
END_IF
END_METHOD

METHOD Init : e_progress
VAR_INPUT
END_VAR
// check pointer and interface
IF NOT Check() THEN Init := e_progress.PROGRESS_ERROR; RETURN; END_IF



// clear all station data
_bInitList                        := _ItfStation^[_nStationId].InitList();

// clear all states and list entries on request
memset(ADR(_stStationCtrl),  0, SIZEOF(_stStationCtrl));
memset(ADR(_stStationState), 0, SIZEOF(_stStationState));

_stStationState.nMask             := 0;
_stStationState.nMoverId          := 0;

_eFatalError                      := 0;

_stStationState.eState            := E_STATION_STATE.STATION_INIT;
_stState^[_nStationId]            := _stStationState;
_sState                           := TO_STRING(_stStationState.eState);

Init                              := e_progress.PROGRESS_DONE;
END_METHOD

PROPERTY ItfMover : pointer to ARRAY[1..MAX_MOVER] OF I_XtsTransport_Mover
SET
_ItfMover := ItfMover;
END_SET
END_PROPERTY

PROPERTY ItfStations : pointer to ARRAY[1..MAX_STATION] OF I_Station_LinkedList
SET
_ItfStation := ItfStations;
END_SET
END_PROPERTY

METHOD PRIVATE MoveData
// build WorkPos from parameter, static station data and information on mover
_stMoveData.rPos            := TO_REAL(_stParameter^[_nStationId].rPosWait
                             + _stParameter^[_nStationId].rPosStop[_nNest]
                             + _stMoverData.rOffset
                             + _rMoverOffset^[_nStationId][_stMoverData.nMoverId][_nNest]);

_stMoveData.rVelo           := _stParameter^[_nStationId].rVelo;
_stMoveData.rAcc            := _stParameter^[_nStationId].rAccDec;
_stMoveData.rJerk           := _stParameter^[_nStationId].rJerk;
_stMoveData.rGap            := _stParameter^[_nStationId].rGap;

// init method and state
_ItfMover^[_stMoverData.nMoverId].MoveToPosCa(FALSE, _stMoveData);
_eState                     := E_PROGRESS.PROGRESS_INIT;
END_METHOD

PROPERTY Mover : POINTER TO ARRAY[1..MAX_MOVER] OF AXIS_REF;
SET
_Mover := Mover;
END_SET
END_PROPERTY

PROPERTY MoverOffset : POINTER TO ARRAY[1..MAX_STATION]  OF T_NEST_OFFSET
SET
_rMoverOffset := MoverOffset;
END_SET
END_PROPERTY

METHOD PRIVATE MoverOut
VAR_INPUT
END_VAR
// build data for sending mover to target station

// who am I sending?
_stMoverDataSend.nMoverId       := _stStationState.nMoverId;

// get optional information about nests to work
_stMoverDataSend.nMask          := _stStationCtrl.nMask;

// get optional offset
_stMoverDataSend.rOffset        := _stStationCtrl.rOffset;

// get target station
_stMoverDataSend.nTargetStation := _stStationCtrl.nTargetStation;

FOR _ix := 1 TO _stParameter^[_stMoverDataSend.nTargetStation].nConfiguredStopCount
DO
  IF GetBitWord(_stMoverDataSend.nMask, _ix-1)
  THEN
    _nNest                      := _ix;
    EXIT;
  END_IF
END_FOR

// get position of target
_stMoveData.rPos                := TO_REAL(_stParameter^[_stMoverDataSend.nTargetStation].rPosWait);

IF (_stMoveData.rPos - TO_REAL(_Mover^[_stMoverDataSend.nMoverId].NcToPlc.ModuloActPos) < 0)
THEN
  // only forward, never back
  _stMoveData.rPos              := TO_REAL(_stMoveData.rPos 
                                 + _ItfMover^[_stMoverDataSend.nMoverId].RailLength);
END_IF

// init method for sending
_ItfMover^[_stMoverDataSend.nMoverId].SendToModuloPosCa(FALSE, 
                                                  _stMoveData);
END_METHOD

METHOD PUBLIC SetBitWord : WORD
VAR_INPUT
  inVal   : WORD;
  bitNo   : DINT;
END_VAR
VAR
  wConst  : WORD := 1;
END_VAR
SetBitWord := inVal OR SHL( wConst,bitNo MOD 16 );
END_METHOD

PROPERTY State : pointer to ARRAY[1..MAX_STATION] OF ST_STATION_STATE
SET
_stState := State;
END_SET
END_PROPERTY

PROPERTY StationId : uint
GET
StationId := _nStationId;
END_GET
SET
_nStationId := StationId;
END_SET
END_PROPERTY

PROPERTY StationParameter : POINTER TO ARRAY[1..MAX_STATION]  OF ST_STATION_PARAMETER
SET
_stParameter := StationParameter;
END_SET
END_PROPERTY

END_FUNCTION_BLOCK

// ---- XTS/Xpu/fb_Xpu.TcPOU
//---------------------------------------------------------------------------------------------------------------
//
//  HAUD 2023.12.14
//
//  - XTS_TRAINING
//  - example project for setting up transport layer
//
//
//  fb_Xpu
//  - connect XTS_Utility.lib to TcCom
//  - cyclic plausibility checks
//  - cyclic ModuleInfoData
//
//  - connection to TcCom Server for local FB instances
//
//
//  CTRL / STATE --> see proprerties
//  structs for use of function block via mapping
//  cyclic check for new command
//
//  VAR INPUT / OUTPUT --> see properties
//
//---------------------------------------------------------------------------------------------------------------
// This SOFTWARE is provided as an Exemple by THE PROVIDER "as is" and "with all faults." THE PROVIDER makes no 
// representations or warranties of any kind concerning the safety, suitability, lack of viruses, inaccuracies, 
// typographical errors, or other harmful components of this SOFTWARE. There are inherent dangers in the use of 
// any software, and you are solely responsible for determining whether this SOFTWARE is compatible with your 
// equipment and other software installed on your equipment. You are also solely responsible for the protection 
// of your equipment and backup of your data, and THE PROVIDER will not be liable for any damages you may suffer 
// in connection with using, modifying, or distributing this SOFTWARE.
//---------------------------------------------------------------------------------------------------------------
FUNCTION_BLOCK fb_Xpu //IMPLEMENTS I_Xpu
VAR
  _eCheck                     : E_XPU_CHECK;
  _eInit                      : E_XPU_INIT;       // MUST equal INIT_DONE for anything to work

  //-------------------------------------------------------------------------------------------------
  // XTS Environment; ProcessingUnit, Part, Track, Mover
  //  - instances are initialized by getting OTCIDs
  //-------------------------------------------------------------------------------------------------
  _nXpu                       : UINT := 1;  // input property in case of multiple XPU in project
  _nGroup                     : UINT;       // input property in case of multiple Xpu in project

  _nTrack                     : UINT := 1;  // this example is intended for one track only

  {attribute 'displaymode':='hex'}
  _CaGroupOID                 : OTCID; // input property frome cyclic CA group interface, MUST be set in order to do successful INIT

  // checked and evaluated in XpuCheckCycle()
  _bAllPositionsValid,
  _bMoverIdDetectionValid,
  _bMoverIdDetectionError     : BOOL;

  _nDetectedMoverCount,
  _nExpectedMoverCount        : UINT;

  _XpuOperationMode           : OperationMode;
  _MoverIdDetectionMode       : MoverIdDetectionMode;

  // XTS_Utility connection to TcCOM Object
  _fbEnvironment              : Tc3_XTS_Utility.FB_TcIoXtsEnvironment;

  // local instances of members of Environment
  // local members are connected to TcCOM by XpuInit()
  _fbProcessingUnit           : Tc3_XTS_Utility.FB_TcIoXtsProcessingUnit;

  _fbXpuPart                  : Tc3_XTS_Utility.FB_TcIoXtsXpuPart;
  _fbXpuTrack                 : Tc3_XTS_Utility.FB_TcIoXtsXpuTrack;

  _fbMc2CaGroup               : Tc3_XTS_Utility.FB_Mc2CaGroup;

  _fbPartModules              : ARRAY[1..MAX_MODULE]  OF Tc3_XTS_Utility.FB_TcIoXtsPartModule;
  _fbMoverXpu                 : ARRAY[1..MAX_MOVER]   OF Tc3_XTS_Utility.FB_TcIoXtsXpuMover;

  // TcCOM ObjectId (who am I talking to?)
  {attribute 'displaymode':='hex'}
  _Xpu_OTCID                  : OTCID;
  {attribute 'displaymode':='hex'}
  _Group_OTCID                : ARRAY[1..MAX_GROUP]   OF OTCID; // OTCID read from XPU
  {attribute 'displaymode':='hex'}
  _Part_OTCID                 : ARRAY[1..MAX_PART]    OF OTCID;
  {attribute 'displaymode':='hex'}
  _Track_OTCID                : ARRAY[1..MAX_TRACK]   OF OTCID;
  {attribute 'displaymode':='hex'}
  _Mov_OTCID                  : ARRAY[1..MAX_MOVER]   OF OTCID;
  {attribute 'displaymode':='hex'}
  _Module_OTCID               : ARRAY[1..MAX_MODULE]  OF OTCID;

  // COE Data access
  _ModuleInfoData             : REFERENCE TO ARRAY[1..MAX_MODULE] OF Tc3_XTS_Utility.ST_InfoDataView;
  _bModulePower               : ARRAY[1..MAX_MODULE] OF BOOL;

  // double check RailLength, XpuInit() will get stuck in error if not configured correctly
  _RailLengthXpu              : LREAL;
  _RailLengthGroup            : LREAL;

  _nLengthXpu,
  _nLengthGroup               : UINT;

  _nInfoServerCount,
  _nIfoStationCount,
  _nPartCount,
  _nTrackCount,
  _nTaskCount,
  _nMoverCount,
  _nModuleCount,
  _nCheckMovOID,
  _nCheckModAdr               : UINT;

  _ix                         : UINT;

  {attribute 'hide'}
  _XpuInfo                    : ST_XPU_INFO;
END_VAR

// get DcLink information from motor modules
PROPERTY AllModulesDcLink : bool
GET
VAR
  _bTmp     : BOOL;
  _nModule  : UINT;
END_VAR
IF NOT (_eInit = E_XPU_INIT.INIT_DONE) THEN RETURN; END_IF

FOR _nModule := 1 TO _nModuleCount
DO
  IF NOT _bModulePower[_nModule] // information comes from cyclic call in Cycle(): ModuleInfoData()
  THEN
    _bTmp  := FALSE;
    EXIT;
  ELSE
    _bTmp  := TRUE;
  END_IF
END_FOR

AllModulesDcLink := _bTmp;
END_GET
END_PROPERTY

PROPERTY CaGroupOID : OTCID
SET
// Group OTCID must come from the CA Group mapping in NC.Objects
_CaGroupOID := CaGroupOID;
END_SET
END_PROPERTY

METHOD Cycle : E_PROGRESS
VAR_INPUT
  Enable      : BOOL; // enable to do cyclic checks on Environment and its members
END_VAR
VAR_IN_OUT
  _eChk       : E_XPU_CHECK;
END_VAR
VAR_INST

  _eJobResult,
  _eResult      : E_PROGRESS;
  _eState       : E_PROGRESS := E_PROGRESS.PROGRESS_INIT;

END_VAR
IF NOT Enable
THEN
  ModuleInfoData(FALSE);

  _eResult  :=
  _eState   := E_PROGRESS.PROGRESS_INIT; 
  _eChk     := E_XPU_CHECK.INIT_CHECK;
END_IF 
//-----------------------------------------------------------------------------
// cyclic data fetch from Environment, ProcessingUnit, Part, ...
//-----------------------------------------------------------------------------
CASE _eState
OF
  E_PROGRESS.PROGRESS_INIT:
    IF Enable
    THEN
      _eState := _eResult         := E_PROGRESS.PROGRESS_BUSY;
    END_IF

  //---------------------------------------------------------------------------
  E_PROGRESS.PROGRESS_BUSY:       // get data from Xpu, ProcessingUnit, Part, XpuCaGroup
    _eState                       := E_PROGRESS.PROGRESS_STARTUP;

    _bAllPositionsValid           := _fbProcessingUnit.GetAreAllPositionsValid();
    _nDetectedMoverCount          := TO_UINT(_fbProcessingUnit.GetDetectedMoverCount());
    _nExpectedMoverCount          := TO_UINT(_fbProcessingUnit.GetExpectedMoverCount());
  
    _XpuOperationMode             := _fbProcessingUnit.GetOperationMode();
    _MoverIdDetectionMode         := _fbProcessingUnit.GetMoverIdDetectionMode();
  
    _RailLengthXpu                := _fbXpuPart.GetLength();
    _RailLengthGroup              := _fbMc2CaGroup.GetRailLength();
    _nLengthXpu                   := TO_UINT(_RailLengthXpu);
    _nLengthGroup                 := TO_UINT(_RailLengthGroup);
END_CASE
//-----------------------------------------------------------------------------
//-----------------------------------------------------------------------------
CASE _eState
OF
  //---------------------------------------------------------------------------
  E_PROGRESS.PROGRESS_STARTUP:    // check data for errors
    IF NOT (_bAllPositionsValid)
    THEN
      _eChk                       := E_XPU_CHECK.PROCESSING_UNIT_POSITIONS_VALID;
      _eState := _eResult         := E_PROGRESS.PROGRESS_ERROR;

    ELSIF NOT (_nLengthXpu > 0)
    THEN
      _eChk                       := E_XPU_CHECK.XPU_RAIL_LENGTH;
      _eState := _eResult         := E_PROGRESS.PROGRESS_ERROR;

    ELSIF NOT (_nLengthGroup > 0)
    THEN
      _eChk                       := E_XPU_CHECK.GROUP_RAIL_LENGTH;
      _eState := _eResult         := E_PROGRESS.PROGRESS_ERROR;
     
    ELSIF NOT (_nDetectedMoverCount = _nExpectedMoverCount)
    THEN
      _bMoverIdDetectionValid     := FALSE;
      _eChk                       := E_XPU_CHECK.MOVER_COUNT_NOT_EQUAL;
      _eState := _eResult         := E_PROGRESS.PROGRESS_ERROR;
  
    ELSIF NOT (_nLengthXpu = _nLengthGroup)
    THEN
      _eChk                       := E_XPU_CHECK.RAIL_LENGTH_COMPARE;
      _eState := _eResult         := E_PROGRESS.PROGRESS_ERROR;
 
    ELSE
      _eResult                    := E_PROGRESS.PROGRESS_WORKING;

      IF NOT (__ISVALIDREF(_ModuleInfoData))
      THEN
        _eState                   := E_PROGRESS.PROGRESS_BUSY;
      ELSE
        _eJobResult               := ModuleInfoData(TRUE);
  
        IF (_eJobResult = E_PROGRESS.PROGRESS_DONE)
        THEN
          _eState                 := E_PROGRESS.PROGRESS_BUSY;
        END_IF  
      END_IF
    END_IF
END_CASE

Cycle                             := _eResult;
END_METHOD

METHOD GetEnvironment : I_TcIoXtsEnvironment
VAR_INPUT
END_VAR
GetEnvironment := _fbEnvironment;
END_METHOD

// mothers' little helper for display in visu
METHOD IdDetectionModeToString : string(20)
VAR
  _DetectionMode    : MoverIdDetectionMode; // Mover ID detection procedure
END_VAR
// just a little helper for visu display
IF NOT (_eInit = E_XPU_INIT.INIT_DONE) THEN IdDetectionModeToString := 'INIT required'; RETURN; END_IF

_DetectionMode := _fbProcessingUnit.GetMoverIdDetectionMode();

CASE _DetectionMode
OF
  MoverIdDetectionMode.Standard:
    IdDetectionModeToString       := 'Standard';

  MoverIdDetectionMode.Mover1:
    IdDetectionModeToString       := 'Mover 1';

  MoverIdDetectionMode.MultipleMover1:
    IdDetectionModeToString       := 'Multiple Mover 1';

ELSE
    IdDetectionModeToString       := 'UNKNOWN Mode';
END_CASE
END_METHOD

// mothers' little helper for display in visu
METHOD ModuleInfoData : E_PROGRESS
VAR_INPUT
  Enable        : BOOL; // enable to read ST_InfoDataView for diag/display
END_VAR
VAR_INST
  _idt,
  _nModule : UINT;
  _eReturn,
  _eState       : E_PROGRESS;
  _aPcbTemp     : ARRAY[1..4] OF REAL;
END_VAR
//---------------------------------------------------------------------------------------------
// just a little helper for visu display
// collects module data for local data
//---------------------------------------------------------------------------------------------
IF NOT (_eInit = E_XPU_INIT.INIT_DONE)      // if Xpu init is not done, just leave
THEN 
  RETURN; 
END_IF
//---------------------------------------------------------------------------------------------
IF NOT Enable                               // clear states on request
THEN
  _eReturn                                  := 
  _eState                                   := E_PROGRESS.PROGRESS_INIT; 
END_IF 
//---------------------------------------------------------------------------------------------
IF NOT (__ISVALIDREF(_ModuleInfoData))      // datafield not connected, error and leave
THEN
  ModuleInfoData                            := E_PROGRESS.PROGRESS_ERROR;
  RETURN;
END_IF
//---------------------------------------------------------------------------------------------
CASE _eState                                // get InfoData from motor modules
OF
  //-------------------------------------------------------------------------------------------
  E_PROGRESS.PROGRESS_INIT:
    IF Enable
    THEN
      _eState                                             := E_PROGRESS.PROGRESS_BUSY;
      _nModule                                            := 1;
    END_IF
END_CASE
CASE _eState
OF
  //-------------------------------------------------------------------------------------------
  E_PROGRESS.PROGRESS_BUSY:
    _eState                                               := E_PROGRESS.PROGRESS_PREPARE;

    _ModuleInfoData[_nModule].fAuxiliaryVoltage_5V        := _fbPartModules[_nModule].GetAuxiliaryVoltage5V();
    _ModuleInfoData[_nModule].fAuxiliaryVoltage_10V       := _fbPartModules[_nModule].GetAuxiliaryVoltage10V();
    _ModuleInfoData[_nModule].fAuxiliaryVoltage_24V       := _fbPartModules[_nModule].GetAuxiliaryVoltage24V();

    _ModuleInfoData[_nModule].fDcLinkVoltage              := _fbPartModules[_nModule].GetDCLinkVoltage();

    IF (_ModuleInfoData[_nModule].fDcLinkVoltage > 48.0*0.85) AND
       (_ModuleInfoData[_nModule].fDcLinkVoltage < 48.0*1.15)
    THEN
      _bModulePower[_nModule]                             := TRUE;
    ELSE
      _bModulePower[_nModule]                             := SEL((_XpuOperationMode = OperationMode.Simulation), FALSE, TRUE);
    END_IF

    _ModuleInfoData[_nModule].nCurrentScaling             := TO_INT(_fbPartModules[_nModule].GetCurrentScaling());

    _ModuleInfoData[_nModule].nDeviceInfo                 := _fbPartModules[_nModule].GetDeviceInfo();

    IF (_XpuOperationMode = OperationMode.Normal)
    THEN
      _ModuleInfoData[_nModule].fAverageTemp              := 0.0;
  
      _aPcbTemp                                           := _fbPartModules[_nModule].GetPCBTemperatures();
  
      _ModuleInfoData[_nModule].fPcbTemp_0                := _aPcbTemp[1];
      _ModuleInfoData[_nModule].fPcbTemp_1                := _aPcbTemp[2];
      _ModuleInfoData[_nModule].fPcbTemp_2                := _aPcbTemp[3];
      _ModuleInfoData[_nModule].fPcbTemp_3                := _aPcbTemp[4];

      FOR _idt := 1 TO 4
      DO
        _ModuleInfoData[_nModule].fAverageTemp            := _ModuleInfoData[_nModule].fAverageTemp + _aPcbTemp[_idt];
      END_FOR
      _ModuleInfoData[_nModule].fAverageTemp              := _ModuleInfoData[_nModule].fAverageTemp / 4;
    END_IF

    _ModuleInfoData[_nModule].fOverallCurrent             := _fbPartModules[_nModule].GetOverallCurrent();

    _ModuleInfoData[_nModule].fMaxDCLinkVoltageLast500ms  := _fbPartModules[_nModule].GetMaxDCLinkVoltageLast500ms();
    _ModuleInfoData[_nModule].fMaxOverallCurrentLast500ms := _fbPartModules[_nModule].GetMaxOverallCurrentLast500ms();
END_CASE
CASE _eState 
OF
  //-------------------------------------------------------------------------------------------
  E_PROGRESS.PROGRESS_PREPARE:
    IF (_nModule > _nModuleCount-1)
    THEN
      _eState                                             := E_PROGRESS.PROGRESS_WORKING;
    ELSE
      _nModule                                            := _nModule + 1;
      _eReturn                                            :=
      _eState                                             := E_PROGRESS.PROGRESS_BUSY;
    END_IF

  //-------------------------------------------------------------------------------------------
  E_PROGRESS.PROGRESS_WORKING:
    _eReturn                                              := E_PROGRESS.PROGRESS_DONE;
    _eState                                               := E_PROGRESS.PROGRESS_INIT;
END_CASE

ModuleInfoData                                            := _eReturn;
END_METHOD

// mothers' little helper for display in visu
METHOD MoverPositionAssignementToString : string(20)
VAR
  _PositionAssignement    : MoverPositionAssignment; // XPU movver assignement procedure
END_VAR
// just a little helper for visu display
IF NOT (_eInit = E_XPU_INIT.INIT_DONE) THEN MoverPositionAssignementToString := 'INIT required'; RETURN; END_IF

_PositionAssignement      := _fbProcessingUnit.GetMoverPositionAssignment();

CASE _PositionAssignement
OF
  MoverPositionAssignment.Standard:
    MoverPositionAssignementToString    := 'Standard';

  MoverPositionAssignment.StartAtFirstMover:
    MoverPositionAssignementToString    := 'Start At First Mover';
ELSE
    MoverPositionAssignementToString    := 'UNKNOWN Assgnement';
END_CASE
END_METHOD

// mothers' little helper for display in visu
METHOD OpModeToString : String(20)
VAR
  _OpMode     : OperationMode; // XPU operation mode
END_VAR
// just a little helper for visu display
IF NOT (_eInit = E_XPU_INIT.INIT_DONE) THEN OpModeToString := 'INIT required'; RETURN; END_IF

_OpMode   := _fbProcessingUnit.GetOperationMode();

CASE _OpMode
OF
  OperationMode.Normal:
    OpModeToString      := 'Normal';

  OperationMode.Simulation:
    OpModeToString      := 'Simulation';

ELSE
    OpModeToString      := 'UNKNOWN OP MODE';
END_CASE
END_METHOD

PROPERTY RailLength : lreal
GET
IF (_eInit = E_XPU_INIT.INIT_DONE)
THEN
  RailLength := _fbXpuPart.GetLength();
ELSE
  RailLength := 0.0;
END_IF
END_GET
END_PROPERTY

PROPERTY XpuInfo : st_xpu_info
GET
IF NOT (_eInit = E_XPU_INIT.INIT_DONE) THEN RETURN; END_IF

_XpuInfo.AllPositionsValid        := _bAllPositionsValid;

_XpuInfo.IdDetectionError         := _bMoverIdDetectionError;
_XpuInfo.IdDetectionValid         := _bMoverIdDetectionValid;

_XpuInfo.IdDetectionActive        := _fbProcessingUnit.GetIsMoverIdDetectionActive();

_XpuInfo.OperationMode            := TO_UINT(_fbProcessingUnit.GetOperationMode());

_XpuInfo.IdDetectionMode          := TO_UINT(_fbProcessingUnit.GetMoverIdDetectionMode());
_XpuInfo.MoverPositionAssignement := TO_UINT(_fbProcessingUnit.GetMoverPositionAssignment());

_XpuInfo.nDetectedAxisCount       := _nDetectedMoverCount;
_XpuInfo.nExpectedAxisCount       := _nExpectedMoverCount;

XpuInfo := _XpuInfo;
END_GET
END_PROPERTY

METHOD XpuInit  : E_XPU_INIT      // connect to TcCOM
VAR_INPUT
  Execute       : BOOL;           // must be executed for connecting to TcCOM Environment of Xpu
END_VAR
VAR_IN_OUT
  _eReslt       : E_PROGRESS;     // send info about progress to caller
  _eChk         : E_XPU_CHECK;
END_VAR
VAR_INST
  _eState         : E_PROGRESS;   // progress state
  _nState         : E_XPU_INIT;   // initialization state
  _eDataGetCount  : E_PROGRESS;   // cycle counter to catch exceeding wait time for data from ProcessingUnit
END_VAR
// clear progress on request
IF NOT Execute 
THEN 
  _eState                           := E_PROGRESS.PROGRESS_INIT;
  _eDataGetCount                    := 0;
 
  XpuInit                           :=
  _nState                           := E_XPU_INIT.INIT_START; 
  RETURN; 
END_IF

// progress state
CASE _eState
OF
  E_PROGRESS.PROGRESS_INIT:         // clear start
    IF Execute
    THEN
      _eState                       := E_PROGRESS.PROGRESS_BUSY;
      _eChk                         := E_XPU_CHECK.INIT_CHECK;    // clear cyclic check state

      // always initialize environment function blocks to get defined start of progress
      _fbEnvironment.Init(FALSE);
      _fbEnvironment.GetXpuOids(FALSE);
      _fbEnvironment.GetInfoServerOids(FALSE);

      // clear initialization states
      _nState                       := E_XPU_INIT.INIT_START;

      // clear check bits
      _bAllPositionsValid           :=
      _bMoverIdDetectionValid       :=
      _bMoverIdDetectionError       := FALSE;

      // clear check values
      _nLengthXpu                   :=
      _nLengthGroup                 :=
      _nDetectedMoverCount          :=
      _nExpectedMoverCount          := 0;

      // clear work values
      _nInfoServerCount             :=
      _nIfoStationCount             :=
      _nPartCount                   :=
      _nTrackCount                  :=
      _nTaskCount                   :=
      _nMoverCount                  :=
      _nModuleCount                 :=
      _nCheckMovOID                 :=
      _nCheckModAdr                 := 0;
    END_IF
END_CASE
//-----------------------------------------------------------------------------
//-----------------------------------------------------------------------------
CASE _eState
OF
  E_PROGRESS.PROGRESS_BUSY:         // begin with initializing environment
    CASE _nState
    OF
    INIT_START:                     // call initialization of environment
      _fbEnvironment.Init(TRUE);

      // get information about success in Property (P_<function>)
      IF _fbEnvironment.P_IsInitialized
      THEN
        // now environment is fully initialized
        // access to members by use of provided interfaces
        // if you use interfaces, things are done here (change to your needs.., rewrite this section...)
        //------------------------------------------------------------------------------------------------
        
        //---------------------------------------------------------------------
        // use of local function block instances
        // get information about Object IDs to local datafields
        //---------------------------------------------------------------------
        //  - everything else in this state machine is for use within fb_Xpu
        //  - the following states shall illustrate how TcCOM Objects are connected through XTS_Utility lib
        //  - local instances of members of Environment are connected from here onward
        //
        IF _fbEnvironment.GetXpuOids(TRUE) // get object IDs for all processing units
        THEN
          _fbEnvironment.Init(FALSE);// clear environment init
          _nState                   := INIT_ENVIRONMENT_OID;
        END_IF
      END_IF

    INIT_ENVIRONMENT_OID:           // get processing unit object ID for THIS instance
      _Xpu_OTCID                    := _fbEnvironment.P_XpuOids[_nXpu];   // fb_Xpu.XpuInstance --> _nXpu

      // clear all local object IDs
      memset(ADR(_Part_OTCID)    , 0, SIZEOF(_Part_OTCID));
      memset(ADR(_Track_OTCID)   , 0, SIZEOF(_Track_OTCID));
      memset(ADR(_Mov_OTCID)     , 0, SIZEOF(_Mov_OTCID));
      memset(ADR(_Module_OTCID)  , 0, SIZEOF(_Module_OTCID));

      // clear function blocks
      _fbEnvironment.GetXpuOids     (FALSE);
      _fbEnvironment.GetCaGroupCount(FALSE);
      _fbEnvironment.GetInfoServerCount(FALSE);

      _nState                       := INIT_INFO_SERVER_ITF;              // check environment for info servers

    INIT_INFO_SERVER_ITF:           // HAUD 2024 03 14: TODO - implement procedure for getting Info server data to local datafields
      IF _fbEnvironment.GetInfoServerCount(TRUE)
      THEN
        // how many of you are there?
        _nInfoServerCount           := _fbEnvironment.P_InfoServerCount;

        IF (_nInfoServerCount > 0)
        THEN
          // go do something with the data
          //
          //  TODO - get station coordinates
          _eState                   := E_PROGRESS.PROGRESS_PREPARE; // TODO - implement InfoServer R/W
          _nState                   := INIT_CA_GROUP_OID;           // TODO - implement initialization states for info server procedure

        ELSE
          // no info server present
          _eState                   := E_PROGRESS.PROGRESS_PREPARE;
          _nState                   := INIT_CA_GROUP_OID; // go check CA group
        END_IF
      END_IF
    END_CASE
END_CASE
//-----------------------------------------------------------------------------
//-----------------------------------------------------------------------------
CASE _eState
OF
  E_PROGRESS.PROGRESS_PREPARE:      // CA group initialization
    CASE _nState
    OF
    INIT_CA_GROUP_OID:              // get object IDs of all CA groups in environment
      IF _fbEnvironment.GetCaGroupOids(TRUE)
      THEN
        _Group_OTCID                := _fbEnvironment.P_CaGroupOids;  // copy all Ids to local
        _nState                     := INIT_CA_GROUP_GET_OID;
      END_IF

    INIT_CA_GROUP_GET_OID:          // look for any CA group
      _fbEnvironment.GetCaGroupOids(FALSE);
      IF NOT (_Group_OTCID[1] <> 0)
      THEN
        // no group is configured in project --> error, go add/link CA Group in NC objects
        _eChk                       := E_XPU_CHECK.GROUP_NOT_CONFIGURED;
        _eState                     := E_PROGRESS.PROGRESS_ERROR;
      ELSE
        _nState                     := INIT_CA_GROUP_CHECK_OID; // get matching CA group
      END_IF

    INIT_CA_GROUP_CHECK_OID:        // ID must be found, there is one chance
      _eChk                         := E_XPU_CHECK.GROUP_OID_MISMATCH;
      _eState                       := E_PROGRESS.PROGRESS_ERROR;

      FOR _ix := 1 TO MAX_GROUP
      DO
        IF (_fbEnvironment.P_CaGroupOids[_ix] <> 0)
        THEN
          // check whether the input from cyclic interface can be found in XPU data
          IF (_fbEnvironment.P_CaGroupOids[_ix] = _CaGroupOID)  // _CaGroupOID must be linked from NC Objects into PLC (GROUP_REF)
          THEN

            _eState                 := E_PROGRESS.PROGRESS_PREPARE;
            _eChk                   := E_XPU_CHECK.INIT_CHECK;

            _nGroup                 := _ix;

            _fbEnvironment.GetCaGroupOids(FALSE);
            _nState                 := INIT_CA_GROUP_COM; // only continue if match was found
            EXIT;
          END_IF
        END_IF
      END_FOR

    INIT_CA_GROUP_COM:              // connect to CaGroup function block in environment
      IF (_fbMc2CaGroup.GetComObject(_fbEnvironment.P_CaGroupOids[_nGroup]))
      THEN
        _eState                     := E_PROGRESS.PROGRESS_STARTUP;
        _nState                     := INIT_PROCESSING_UNIT_COM;
      END_IF
    END_CASE
END_CASE
//-----------------------------------------------------------------------------
//-----------------------------------------------------------------------------
CASE _eState
OF
  E_PROGRESS.PROGRESS_STARTUP:      // ProcessingUnit initialization
  CASE _nState
  OF
  INIT_PROCESSING_UNIT_COM:         // connect local function block with TcCom object
    IF (_fbProcessingUnit.GetComObject(_Xpu_OTCID))
    THEN
      // local function block can now be used to get information
      // get operation mode first
      _XpuOperationMode             := _fbProcessingUnit.GetOperationMode();
      _nState                       := INIT_PROCESSING_UNIT_PART_COUNT;
    END_IF

  INIT_PROCESSING_UNIT_PART_COUNT:  // get parts in ProcessingUnit
    _nPartCount                     := TO_UINT(_fbProcessingUnit.GetPartCount());

    IF (_nPartCount > 0)            // one is enough
    THEN
      _nState                       := INIT_PROCESSING_UNIT_PART_OID;
    END_IF

  INIT_PROCESSING_UNIT_PART_OID:    // get object IDs of all parts in ProcessingUNit
    IF _fbProcessingUnit.GetPartOids()
    THEN
      _eState                       := E_PROGRESS.PROGRESS_CHECK;

      _Part_OTCID                   := _fbProcessingUnit.P_PartOids;  // copy IDs to local
      _nState                       := INIT_PROCESSING_UNIT_TRACK_COUNT;
    END_IF
  END_CASE
END_CASE
//-----------------------------------------------------------------------------
//-----------------------------------------------------------------------------
CASE _eState
OF
  E_PROGRESS.PROGRESS_CHECK:        // track initialization
  CASE _nState
  OF
  INIT_PROCESSING_UNIT_TRACK_COUNT: // how many tracks does this ProcessingUnit have?
    _nTrackCount                    := TO_UINT(_fbProcessingUnit.GetTrackCount());
  
    IF (_nTrackCount > 0)           // one is enough
    THEN
      _nState                       := INIT_PROCESSING_UNIT_TRACK_OID;
    END_IF

  INIT_PROCESSING_UNIT_TRACK_OID:   // get object IDs of all tracks in ProcessingUnit
    IF _fbProcessingUnit.GetTrackOids()
    THEN
      _eState                       := E_PROGRESS.PROGRESS_OCCUPIED;

      _Track_OTCID                  := _fbProcessingUnit.P_TrackOids; // copy IDs to local
      _nState                       := INIT_PROCESSING_UNIT_MOVER_COUNT;
    END_IF
  END_CASE
END_CASE
//-----------------------------------------------------------------------------
//-----------------------------------------------------------------------------
CASE _eState
OF
  E_PROGRESS.PROGRESS_OCCUPIED:     // Mover initialization
  CASE _nState
  OF
  INIT_PROCESSING_UNIT_MOVER_COUNT: // how many of you are there?
    _nMoverCount                    := TO_UINT(_fbProcessingUnit.GetMoverCount());
  
    IF (_nMoverCount > 0)           // one is enough
    THEN
      _nState                       := INIT_PROCESSING_UNIT_MOVER_OID;
    END_IF

  INIT_PROCESSING_UNIT_MOVER_OID:   // get object IDs of all mover in ProcessingUnit
    IF _fbProcessingUnit.GetMoverOids()
    THEN
      _eState                       := E_PROGRESS.PROGRESS_WORKING;

      _Mov_OTCID                    := _fbProcessingUnit.P_MoverOids; // copy IDs to local
      _nState                       := INIT_PROCESSING_UNIT_TASK_COUNT;
      _eChk                         := E_XPU_CHECK.MOVER_COUNT;
    END_IF
  END_CASE
END_CASE
//-----------------------------------------------------------------------------
//-----------------------------------------------------------------------------
CASE _eState
OF
  E_PROGRESS.PROGRESS_WORKING:      // task information
  CASE _nState
  OF
  INIT_PROCESSING_UNIT_TASK_COUNT:  // how many?
    _nTaskCount                     := TO_UINT(_fbProcessingUnit.GetTaskCount());
  
    IF (_nTaskCount > 0)
    THEN
      _nState                       := INIT_PROCESSING_UNIT_TASK_OID;
    END_IF    

  INIT_PROCESSING_UNIT_TASK_OID:    // get their names!
    IF _fbProcessingUnit.GetTaskOids()
    THEN
      _eState                       := E_PROGRESS.PROGRESS_STILL_WORKING;
      _nState                       := INIT_TRACK_COM;
    END_IF
  END_CASE
END_CASE
//-----------------------------------------------------------------------------
//-----------------------------------------------------------------------------
CASE _eState
OF
  E_PROGRESS.PROGRESS_STILL_WORKING:// connect local instances of track, part, modules and mover
    CASE _nState
    OF
    INIT_TRACK_COM:                 // get TcCom Object for my track (_nTrack is fixed to 1 in this example; multi track is not intended)
      IF _fbXpuTrack.GetComObject(_Track_OTCID[_nTrack])
      THEN
        _nState                     := INIT_PART_COM;
      END_IF
    //-----------------------------------------------------------------------------------------------
    //-----------------------------------------------------------------------------------------------
    INIT_PART_COM:                  // get TcCom object for my part (also fixed to 1 part per ProcessingUnit; multi part is not intended)
      IF _fbXpuPart.GetComObject(_Part_OTCID[1])
      THEN
        _nState                     := INIT_PART_MODULE_COUNT;
      END_IF
    //-----------------------------------------------------------------------------------------------
    //-----------------------------------------------------------------------------------------------
    INIT_PART_MODULE_COUNT:         // get count of motor modules
      _nModuleCount                 := TO_UINT(_fbXpuPart.GetModuleCount());
    
      IF (_nModuleCount > 0)        // one is enough
      THEN
        _nState                     := INIT_PART_MODULE_OID;
      END_IF
    //-----------------------------------------------------------------------------------------------
    //-----------------------------------------------------------------------------------------------
    INIT_PART_MODULE_OID:           // get object IDs of all motor modules in part
      IF _fbXpuPart.GetModuleOids()
      THEN
        _Module_OTCID               := _fbXpuPart.P_ModuleOids; // copy IDs to local
    
        _nState                     := INIT_PART_MODULE_COM;    // go, connect module IDs
        _nCheckModAdr               := 1;                       // start at first module
      END_IF
    //-----------------------------------------------------------------------------------------------
    //-----------------------------------------------------------------------------------------------
    INIT_PART_MODULE_COM:           // connect to TcCom object
      IF _fbPartModules[_nCheckModAdr].GetComObject(_Module_OTCID[_nCheckModAdr])
      THEN
        _nState                     := INIT_PART_MODULE_COM_NEXT;
      END_IF
    //-----------------------------------------------------------------------------------------------
    INIT_PART_MODULE_COM_NEXT:
      IF (_nCheckModAdr > _nModuleCount-1)
      THEN
        // all data from modules collected, continue to mover data
        _nState                     := INIT_MOVER_COM;          // go, connect mover IDs 
        _nCheckMovOID               :=  1;                      // start at first mover
      ELSE
        // still data to fetch, increment search index, go back to fetching data
        _nState                     := INIT_PART_MODULE_COM;    // go back for next
        _nCheckModAdr               := _nCheckModAdr + 1;       // next
      END_IF
    //-----------------------------------------------------------------------------------------------
    //-----------------------------------------------------------------------------------------------
    INIT_MOVER_COM:                 // connect to TcCom object
      IF _fbMoverXpu[_nCheckMovOID].GetComObject(_Mov_OTCID[_nCheckMovOID])
      THEN
        _nState                     := INIT_MOVER_COM_NEXT;
      END_IF
    //-----------------------------------------------------------------------------------------------
    INIT_MOVER_COM_NEXT:
      IF (_nCheckMovOID > _nMoverCount-1)
      THEN
        // all done
        _nState                     := INIT_DATA_GET;           // get important data from ProcessingUnit etc...
      ELSE
        // more data to fetch, increment search index and go back
        _nState                     := INIT_MOVER_COM;          // go back for next
        _nCheckMovOID               := _nCheckMovOID + 1;       // next
      END_IF
    //-----------------------------------------------------------------------------------------------
    //-----------------------------------------------------------------------------------------------
    INIT_DATA_GET:                  // get data, add more if your application requires it
      // start counter
      _eDataGetCount                := _eDataGetCount + 1;
      IF (_eDataGetCount MOD E_PROGRESS.PROGRESS_ERROR = 0)
      THEN
        _eState                     := E_PROGRESS.PROGRESS_ERROR;
        _eCheck                     := E_XPU_CHECK.PROCESSING_UNIT_GET_DATA_EXCEED;
      END_IF
      // wait for plausible data from members
      IF (_bAllPositionsValid) AND
         (_nLengthXpu > 0)
      THEN
        _nState                     := INIT_DATA_CHECK;
        _eChk                       := E_XPU_CHECK.PROCESSING_UNIT_POSITIONS_VALID;
      END_IF

      _bAllPositionsValid           := _fbProcessingUnit.GetAreAllPositionsValid();
      _nDetectedMoverCount          := TO_UINT(_fbProcessingUnit.GetDetectedMoverCount());
      _nExpectedMoverCount          := TO_UINT(_fbProcessingUnit.GetExpectedMoverCount());

      _XpuOperationMode             := _fbProcessingUnit.GetOperationMode();
      _MoverIdDetectionMode         := _fbProcessingUnit.GetMoverIdDetectionMode();

      _RailLengthXpu                := _fbXpuPart.GetLength();
      _RailLengthGroup              := _fbMc2CaGroup.GetRailLength();
      _nLengthXpu                   := TO_UINT(_RailLengthXpu);
      _nLengthGroup                 := TO_UINT(_RailLengthGroup);

    //-----------------------------------------------------------------------------------------------
    INIT_DATA_CHECK:                // plausibility checks
      IF NOT (_nDetectedMoverCount = _nExpectedMoverCount)
      THEN
        _eChk                       := E_XPU_CHECK.MOVER_COUNT_NOT_EQUAL; // the thing that must not be
        _eState                     := E_PROGRESS.PROGRESS_ERROR;

      ELSIF NOT (_nLengthXpu = _nLengthGroup)
      THEN
        _eChk                       := E_XPU_CHECK.RAIL_LENGTH_COMPARE;   // yet another thing that must not be
        _eState                     := E_PROGRESS.PROGRESS_ERROR;

      ELSE
        _nState                     := INIT_DONE;                         // write success
      END_IF
    //-----------------------------------------------------------------------------------------------
    INIT_DONE:
      _eState                       := E_PROGRESS.PROGRESS_DONE;          // method is done
    END_CASE
END_CASE

_eReslt                             := _eState;
XpuInit                             := _nState;
END_METHOD

PROPERTY XpuInstance : uint
SET
//
// Who am I?
// Environment may have more than one ProcessingUnit,
// information required for connecting to the correct instance of ProcessingUnit
_nXpu := XpuInstance;
END_SET
END_PROPERTY

PROPERTY XpuModuleInfoData : REFERENCE TO ARRAY[1..MAX_MODULE] OF Tc3_XTS_Utility.ST_InfoDataView
SET

_ModuleInfoData REF= XpuModuleInfoData;
END_SET
END_PROPERTY

END_FUNCTION_BLOCK

// ---- XTS/XtsTransportUnit/fb_TransportUnit.TcPOU
//---------------------------------------------------------------------------------------------------------------
//
//  HAUD 2024.03.18
//
//  - XTS_TRAINING
//  - example project for setting up transport layer
//
//
//  fb_TransportUnit
//  - Ctrl/STate interface, reacts to change of command
//  - controls members via structures and interfaces for getting XTS in defined state
//    - Transport Init
//        - XPU is initialized
//        - XPU detects mover
//
//    - Transport Idle
//      - Cyclic Checks of XPU and CaGroup
//
//
//  CTRL / STATE --> see proprerties
//  structs for use of function block via mapping
//  cyclic check for new command
//
//  VAR INPUT / OUTPUT --> see properties
//
//---------------------------------------------------------------------------------------------------------------
// This SOFTWARE is provided as an Exemple by THE PROVIDER "as is" and "with all faults." THE PROVIDER makes no 
// representations or warranties of any kind concerning the safety, suitability, lack of viruses, inaccuracies, 
// typographical errors, or other harmful components of this SOFTWARE. There are inherent dangers in the use of 
// any software, and you are solely responsible for determining whether this SOFTWARE is compatible with your 
// equipment and other software installed on your equipment. You are also solely responsible for the protection 
// of your equipment and backup of your data, and THE PROVIDER will not be liable for any damages you may suffer 
// in connection with using, modifying, or distributing this SOFTWARE.
//---------------------------------------------------------------------------------------------------------------
FUNCTION_BLOCK fb_TransportUnit
VAR
  _eCheck                       : E_XTS_TRANSPORT_CHECK;

  // Transport Ctrl/State
  _Ctrl                         : REFERENCE TO ST_XTS_TRANSPORT_CTRL;
  _State                        : REFERENCE TO ST_XTS_TRANSPORT_STATE;


  // execute transport commands
  _eCmd,
  _eCmdOld                      : E_XTS_TRANSPORT_CTRL;

  // execution state
  _eState                       : E_XTS_TRANSPORT_STATE;

  // execution result
  _eJobResult,
  _eResult                      : E_PROGRESS;


  // members of transport
  _XpuCtrl                      : REFERENCE TO ST_XPU_CTRL;                     // processing unit ctrl
  _XpuState                     : REFERENCE TO ST_XPU_STATE;                    // processing unit state
  _XpuInfo                      : REFERENCE TO ST_XPU_INFO;                     // processing unit information

  _GroupItf                     : I_XtsTransport_CaGroup;                       // group methods
  _GroupInfo                    : REFERENCE TO ST_GROUP_INFO;                   // info from group

  _MoverItf                     : REFERENCE TO ARRAY[1..MAX_MOVER] OF I_XtsTransport_Mover;  // mover methods
  _MoverInfo                    : REFERENCE TO ARRAY[1..MAX_MOVER] OF ST_MOVER_INFO;         // info from mover

  _StationStart                 : REFERENCE TO ST_STATION_PARAMETER;            // position, gap, dynamic constraints for sending all mover to start position

  // stations lists
  _ItfStationList               : REFERENCE TO ARRAY[1..MAX_STATION]  OF I_Station_LinkedList;  // access to all stations lists

  // access to stations methods by interface
  _ItfStationCtrl               : REFERENCE TO ARRAY[1..MAX_STATION]  OF I_XtsTransport_Station;

  _nStartStation                : UINT;

  _stMoverDataSend              : ST_STATION_MOVER_DATA;    // mover ticket data

  _stListResult                 : ST_STATION_LIST_RESULT;
END_VAR

IF NOT Check() THEN RETURN; END_IF

_eCmd                         := _Ctrl.Cmd;

// check for command change
// get state for cmd
IF (_eCmd <> _eCmdOld)
THEN
  _eState                     := Cmd(_eCmd);
  _eCmdOld                    := _eCmd;
END_IF


CASE _eState
OF
  E_XTS_TRANSPORT_STATE.TRANSPORT_INIT:
    _eResult                  := XpuInit(TRUE);

  E_XTS_TRANSPORT_STATE.TRANSPORT_IDLE:
    _eResult                  := f_GetProgress(_XpuState.State);

    IF (_GroupInfo.GroupErrorStop) OR
       (_GroupInfo.GroupError)
    THEN
      _eResult                := E_PROGRESS.PROGRESS_ERROR;
    END_IF

  E_XTS_TRANSPORT_STATE.TRANSPORT_MOVER_ENABLE:
    _eResult                  := MoverEnableAll(TRUE);

  E_XTS_TRANSPORT_STATE.TRANSPORT_MOVER_DISABLE:
    _eResult                  := MoverDisableAll(TRUE);

  E_XTS_TRANSPORT_STATE.TRANSPORT_GROUP_CLEAR:
    _eResult                  := GroupClear(TRUE);

  E_XTS_TRANSPORT_STATE.TRANSPORT_GROUP_BUILD:
    _eResult                  := GroupBuild(TRUE);

  E_XTS_TRANSPORT_STATE.TRANSPORT_GROUP_ENABLE:
    _eResult                  := GroupEnable(TRUE);

  E_XTS_TRANSPORT_STATE.TRANSPORT_START:
    _eResult                  := TransportStart(TRUE);

  E_XTS_TRANSPORT_STATE.TRANSPORT_RESTART:
    _eResult                  := TransportRestart(TRUE);

ELSE
  _eResult                    := E_PROGRESS.PROGRESS_INVALID;
END_CASE


CASE _eResult
OF
  E_PROGRESS.PROGRESS_INVALID:
    _State.State              := TO_UINT(_eResult);

  E_PROGRESS.PROGRESS_ERROR:
    _State.State              := _eState + E_PROGRESS.PROGRESS_ERROR;

  E_PROGRESS.PROGRESS_DONE:
    _State.State              := _eState + E_PROGRESS.PROGRESS_DONE;

ELSE
  _State.State                := _eState + _eResult;
END_CASE

_State.XpuState               := _XpuState;
_State.GroupInfo              := _GroupInfo;

METHOD PRIVATE Check  : BOOL
VAR_INST
  _idx        : UINT;
END_VAR

IF NOT __ISVALIDREF(_Ctrl)
THEN
  _eCheck                     := E_XTS_TRANSPORT_CHECK.POINTER_NULL_CTRL;
  RETURN;
END_IF

IF NOT __ISVALIDREF(_State)
THEN
  _eCheck                     := E_XTS_TRANSPORT_CHECK.POINTER_NULL_STATE;
  RETURN;
END_IF

_State.Check                  := _eCheck;

IF NOT __ISVALIDREF(_XpuCtrl)
THEN
  _eCheck                     := E_XTS_TRANSPORT_CHECK.POINTER_NULL_XPU_CTRL;
  RETURN;
END_IF

IF NOT __ISVALIDREF(_XpuState)
THEN
  _eCheck                     := E_XTS_TRANSPORT_CHECK.POINTER_NULL_XPU_STATE;
  RETURN;
END_IF

IF NOT __ISVALIDREF(_XpuInfo)
THEN
  _eCheck                     := E_XTS_TRANSPORT_CHECK.POINTER_NULL_XPU_INFO;
  RETURN;
END_IF

IF NOT (_GroupItf <> 0)
THEN
  _eCheck                     := E_XTS_TRANSPORT_CHECK.POINTER_NULL_GROUP_ITF;
  RETURN;
END_IF

IF NOT __ISVALIDREF(_GroupInfo)
THEN
  _eCheck                     := E_XTS_TRANSPORT_CHECK.POINTER_NULL_GROUP_INFO;
  RETURN;
END_IF

IF NOT __ISVALIDREF(_MoverItf)
THEN
  _eCheck                     := E_XTS_TRANSPORT_CHECK.POINTER_NULL_MOVER;
  RETURN;
END_IF

FOR _idx := 1 TO MAX_MOVER
DO
  IF NOT (_MoverItf[_idx] <> 0)
  THEN
    _eCheck                   := E_XTS_TRANSPORT_CHECK.POINTER_NULL_MOVER_ITF;
    RETURN;
  END_IF
END_FOR

IF NOT __ISVALIDREF(_MoverInfo)
THEN
  _eCheck                     := E_XTS_TRANSPORT_CHECK.POINTER_NULL_MOVER_INFO;
  RETURN;
END_IF

IF NOT __ISVALIDREF(_StationStart)
THEN
  _eCheck                     := E_XTS_TRANSPORT_CHECK.POINTER_NULL_STATION_START;
  RETURN;
END_IF

IF NOT __ISVALIDREF(_ItfStationList)
THEN
  _eCheck                     := E_XTS_TRANSPORT_CHECK.POINTER_NULL_STATION_ITF;
  RETURN;
END_IF

IF NOT __ISVALIDREF(_ItfStationCtrl)
THEN
  _eCheck                     := E_XTS_TRANSPORT_CHECK.POINTER_NULL_STATION_CTRL;
  RETURN;
END_IF


_eCheck                       := E_XTS_TRANSPORT_CHECK.DONE_CHECK;
Check                         := TRUE;
END_METHOD

METHOD PRIVATE Cmd : E_XTS_TRANSPORT_STATE
VAR_INPUT
  Ctrl      : E_XTS_TRANSPORT_CTRL;
END_VAR
VAR_INST
  _eRslt    : E_PROGRESS;
  _eState   : E_XTS_TRANSPORT_STATE;
  _eCk      : E_XTS_TRANSPORT_CHECK;
END_VAR
IF NOT Check() THEN RETURN; END_IF


CASE Ctrl
OF
  E_XTS_TRANSPORT_CTRL.CMD_NULL:  // clear all method calls
    _eState               := E_XTS_TRANSPORT_STATE.TRANSPORT_NULL;
    _eRslt                := XpuInit         (FALSE);
    _eRslt                := GroupClear      (FALSE);
    _eRslt                := GroupBuild      (FALSE);
    _eRslt                := GroupEnable     (FALSE);
    _eRslt                := MoverEnableAll  (FALSE);
    _eRslt                := MoverDisableAll (FALSE);
    _eRslt                := TransportRestart(FALSE);
    _eRslt                := TransportRestart(FALSE);

  E_XTS_TRANSPORT_CTRL.CMD_INIT:  // clear methods for initialization
    _eState               := E_XTS_TRANSPORT_STATE.TRANSPORT_INIT;
    _eResult              := XpuInit(FALSE);


ELSE
  IF NOT (_XpuState.Init = E_XPU_INIT.INIT_DONE)
  THEN
    // no init, no further commands possible
    _eState               := E_XTS_TRANSPORT_STATE.TRANSPORT_INVALID;
  ELSE
    CASE Ctrl
    OF
      E_XTS_TRANSPORT_CTRL.CMD_IDLE:
        _eState           := E_XTS_TRANSPORT_STATE.TRANSPORT_IDLE;

      E_XTS_TRANSPORT_CTRL.CMD_MOVER_ENABLE:
        _eState           := E_XTS_TRANSPORT_STATE.TRANSPORT_MOVER_ENABLE;
        _eResult          := MoverEnableAll(FALSE);

      E_XTS_TRANSPORT_CTRL.CMD_MOVER_DISABLE:
        _eState           := E_XTS_TRANSPORT_STATE.TRANSPORT_MOVER_DISABLE;
        _eResult          := MoverDisableAll(FALSE);

      E_XTS_TRANSPORT_CTRL.CMD_GROUP_CLEAR:
        _eState           := E_XTS_TRANSPORT_STATE.TRANSPORT_GROUP_CLEAR;
        _eResult          := GroupClear (FALSE);

      E_XTS_TRANSPORT_CTRL.CMD_GROUP_BUILD:
        _eState           := E_XTS_TRANSPORT_STATE.TRANSPORT_GROUP_BUILD;
        _eResult          := GroupBuild (FALSE);

      E_XTS_TRANSPORT_CTRL.CMD_GROUP_ENABLE:
        _eState           := E_XTS_TRANSPORT_STATE.TRANSPORT_GROUP_ENABLE;
        _eResult          := GroupEnable(FALSE);

      E_XTS_TRANSPORT_CTRL.CMD_TRANSPORT_START:
        _eState           := E_XTS_TRANSPORT_STATE.TRANSPORT_START;
        _eResult          := TransportStart(FALSE);

      E_XTS_TRANSPORT_CTRL.CMD_TRANSPORT_RESTART:
        _eState           := E_XTS_TRANSPORT_STATE.TRANSPORT_RESTART;
        _eResult          := TransportRestart(FALSE);

    ELSE
        _eState           := E_XTS_TRANSPORT_STATE.TRANSPORT_INVALID;
    END_CASE
  END_IF
END_CASE

Cmd                       := _eState;
END_METHOD

PROPERTY Ctrl : REFERENCE TO ST_XTS_TRANSPORT_CTRL
SET
_Ctrl REF= Ctrl;
END_SET
END_PROPERTY

METHOD GroupBuild : E_PROGRESS
VAR_INPUT
  Execute     : BOOL;
END_VAR
VAR_INST
  _nErrorId   : UDINT;
  _eJobReslt,
  _eState     : E_PROGRESS;
END_VAR
//-----------------------------------------------------------------------------
IF NOT Execute 
THEN 
	_eState                       := E_PROGRESS.PROGRESS_INIT; 
END_IF 
//-----------------------------------------------------------------------------
IF NOT Check() 
THEN 
	GroupBuild                    := E_PROGRESS.PROGRESS_ERROR; 
	RETURN; 
END_IF
//-----------------------------------------------------------------------------
//-----------------------------------------------------------------------------
CASE _eState
OF
  E_PROGRESS.PROGRESS_INIT:
    IF Execute
    THEN
      _nErrorId                 := 0;

      IF (_GroupInfo.AxisCount <> 0)
      THEN
        _nErrorId               := 9999;
        _eState                 := E_PROGRESS.PROGRESS_ERROR;
      ELSE
        _eState                 := E_PROGRESS.PROGRESS_BUSY;
        _eJobReslt              := _GroupItf.AddAll(FALSE);
      END_IF
    END_IF
END_CASE
//---------------------------------------------------------------------------
//---------------------------------------------------------------------------
CASE _eState
OF
  E_PROGRESS.PROGRESS_BUSY:
    _eJobReslt                  := _GroupItf.AddAll(TRUE);

    IF (_eJobReslt = E_PROGRESS.PROGRESS_ERROR)
    THEN
      _eState                   := E_PROGRESS.PROGRESS_ERROR;

      _nErrorId                 := _GroupInfo.GroupErrorId;
      _eJobReslt                := _GroupItf.AddAll(FALSE);

    ELSIF (_eJobReslt = E_PROGRESS.PROGRESS_DONE)
    THEN
      _eState                   := E_PROGRESS.PROGRESS_DONE;
      _eJobReslt                := _GroupItf.AddAll(FALSE);
    END_IF
END_CASE
//-----------------------------------------------------------------------------
//-----------------------------------------------------------------------------

GroupBuild                      := _eState;
END_METHOD

